(* CODESYS project mobject-graph.library
   Company: mobject
   DefaultNamespace: mobject-graph
   Version: 0.1.0
   Placeholder: mobject-graph
   Author: mobject dev team
   Title: mobject-graph

Project tree, tasks and I/O mapping:
  libraries: mobject-collections, 1.1.0 (mobject); mobject-datatypes, 0.4.1 (mobject); mobject-deserialization, 0.1.0 (mobject); mobject-disposable, 1.0.0 (mobject); mobject-enumerable, 1.1.0 (mobject); mobject-errors, 0.2.0 (mobject); mobject-events, 1.0.0 (mobject); mobject-serialization, 0.4.0 (mobject); Tc2_Standard, * (Beckhoff Automation GmbH); Tc2_System, * (Beckhoff Automation GmbH); Tc2_Utilities, * (Beckhoff Automation GmbH)
  Alarms/
    Base/
      function block Alarm [ST]: Active, Clear, Message, Reason, FB_init, Accept, RegisterWithParent, SerializeWith
    Events/
      function block AlarmAddedEvent [ST]: FB_init, Target
      interface I_AlarmAddedEvent: Target
    Host/
      function block AlarmHost [ST]: FB_init, EmitOnAlarmAddedEvent, Accept, AddAlarm, HasAlarms, HasRaisedAlarm, SerializeWith
    Interfaces/
      interface I_Alarm: Accept, Active, Message, Reason
      interface I_Alarms: Accept, AddAlarm, HasAlarms, HasRaisedAlarm
      interface I_HostAlarms: Alarms
    function block DeserializationFailedAlarm [ST]: Active, Clear, Message, Raise, Reason
    function block DeserializationFailedNodeNotSupportedAlarm [ST]: Active, Clear, Message, Raise, Reason
    function block FunctionFailedAlarm [ST]: Active, Clear, Message, Raise, Reason
  Content/
    Base/
      function block Content [ST]: FB_init, Accept, AddMetadata, Data, Metadatum, Name, OffEvent, OnceEvent, OnEvent, Parent, RegisterWithParent, SerializeWith
    Events/
      function block ContentAddedEvent [ST]: FB_init, Target
      interface I_ContentAddedEvent: Target
    Host/
      function block ContentHost [ST]: FB_init, FB_exit, CreateContent, DisposeSelfCreatedContent, EmitOnContentAddedEvent, Accept, AddContent, AddDataAsContent, HasContents, SerializeWith, TryGetContentByName
    Interface/
      interface I_Content: Accept, Data, Name, Parent
      interface I_Contents: Accept, AddContent, AddDataAsContent, HasContents, TryGetContentByName
      interface I_HostContent: Contents
  Errors/
    function block MissingNodePrototypeDeserializationError [ST]: FB_init, ErrorType, Message
  Extensions/
    Base/
      function block Extension [ST]: FB_init, Accept, AddMetadata, Alarms, Contents, HasRaisedAlarm, InputPorts, Metadatum, Name, OffEvent, OnceEvent, OnEvent, OutputPorts, Parameters, SerializeWith, TryDeserializeFrom
    Events/
      function block ExtensionAddedEvent [ST]: FB_init, Target
      interface I_ExtensionAddedEvent: Target
    Host/
      function block ExtensionHost [ST]: FB_init, EmitOnExtensionAddedEvent, Accept, AddExtension, HasExtensions, SerializeWith, TryDeserializeFrom, TryGetExtensionByName
    Interface/
      interface I_Extension: Accept, Name
      interface I_Extensions: Accept, AddExtension, HasExtensions, TryGetExtensionByName
      interface I_HostExtensions: Extensions
    Namespace/
      function block ExtensionNamespace [ST]: FB_init, ExtensionName, Initialize, IsExtensionPath, TargetName
  Graph/
    Base/
      function block Graph [ST]: FB_init, FB_exit, DisposeSelfCreatedNodes, TryDeserializeLinks, TryDeserializeNodes, Accept, AddMetadata, Alarms, Contents, Execute, Extensions, HasRaisedAlarm, InputPorts, Metadatum, Nodes, OffEvent, OnceEvent, OnEvent, OutputPorts, Parameters, Reset, SerializeWith, TryDeserializeFrom, Uuid
    Events/
      function block GraphAddedEvent [ST]: FB_init, Target
      interface I_GraphAddedEvent: Target
    Host/
      function block GraphHost [ST]: FB_init, EmitOnGraphAddedEvent, Accept, AddGraph, DisposeAll, Execute, RemoveGraph, SerializeWith, TryGetGraphByUuid
    Interfaces/
      interface I_Graph: Accept, Execute, Reset, Uuid
      interface I_Graphs: Accept, AddGraph, DisposeAll, Execute, RemoveGraph, TryGetGraphByUuid
      interface I_HostGraphs: Graphs
  GraphFramework/
    Interface/
      interface I_GraphFramework: Create, Datatypes, NodeFactory
    function block GraphFramework [ST]: Create, Datatypes, InstallDatatypePack, InstallNodePack, NodeFactory
  InputPort/
    Base/
      function block InputPort [ST]: FB_init, EmitOnInputPortChanged, HandleOutputPortChangedEvent, Accept, AddMetadata, Connected, Data, Disconnect, HandleEvent, Metadatum, Name, OffEvent, OnceEvent, OnEvent, RegisterWithParent, SerializeWith, TryConnectTo
    Events/
      interface I_InputPortAddedEvent: Target
      interface I_InputPortChangedEvent: Target
      function block InputPortAddedEvent [ST]: FB_init, Target
      function block InputPortChangedEvent [ST]: FB_init, Target
    Host/
      function block InputPortHost [ST]: FB_init, FB_exit, CreateInputPort, DisposeSelfCreatedInputPorts, EmitOnPortAddedEvent, Accept, AddDataAsInputPort, AddInputPort, HasInputPorts, SerializeWith, TryGetInputPortByName
    Interface/
      interface I_HostInputPorts: InputPorts
      interface I_InputPort: Accept, Connected, Data, Disconnect, Name, TryConnectTo
      interface I_InputPorts: Accept, AddDataAsInputPort, AddInputPort, HasInputPorts, TryGetInputPortByName
  Metadata/
    Base/
      function block Metadata [ST]: FB_init, Accept, Data, Name, Parent, RegisterWithParent, SerializeWith
    Events/
      interface I_MetadataAddedEvent: Target
      function block MetadataAddedEvent [ST]: FB_init, Target
    Host/
      function block MetadataHost [ST]: FB_init, FB_exit, CreateMetadata, DisposeSelfCreatedMetadata, EmitOnMetadataAddedEvent, Accept, AddDataAsMetadata, AddMetadata, HasMetadata, SerializeWith, TryGetMetadataByName
    Interface/
      interface I_HostMetadata: AddMetadata, Metadatum
      interface I_Metadata: Accept, Data, Name, SerializeWith
      interface I_Metadatum: Accept, AddDataAsMetadata, AddMetadata, HasMetadata, TryGetMetadataByName
  Node/
    Base/
      function block Node [ST]: Clone, OnExecute, EmitNodeExecuteBeginEvent, EmitNodeExecuteEndEvent, EmitOnNodePreExecuteEvent, AddContent, AddInput, AddOutput, AddParameter, Accept, AddMetadata, Alarms, Contents, Execute, Extensions, HasRaisedAlarm, Id, InputPorts, Metadatum, Mode, OffEvent, OnceEvent, OnEvent, Order, OutputPorts, Parameters, Self, SerializeWith, TryDeserializeFrom
    Events/
      interface I_NodeAddedEvent: Target
      interface I_NodeExecuteBeginEvent: Target
      interface I_NodeExecuteEndEvent: Target
      interface I_NodePreExecuteEvent: Cancel, ExecuteCancelled, Target
      function block NodeAddedEvent [ST]: FB_init, Target
      function block NodeExecuteBeginEvent [ST]: FB_init, CpuCounterHighBytes, CpuCounterLowBytes, Target
      function block NodeExecuteEndEvent [ST]: FB_init, CpuCounterHighBytes, CpuCounterLowBytes, Target
      function block NodePreExecuteEvent [ST]: FB_init, Cancel, ExecuteCancelled, Target
    Host/
      function block NodeHost [ST]: FB_init, EmitOnNodeAddedEvent, UpdateExecutionOrder, Accept, AddNode, Execute, HasNodes, RemoveNode, SerializeWith, TryDeserializeFrom, TryGetNodeById
    Interface/
      interface I_HostNodes: Nodes
      interface I_Node: Accept, Clone, Execute, Id, Mode, Order
      interface I_Nodes: Accept, AddNode, HasNodes, TryGetNodeById
  NodeFactory/
    Base/
      function block NodeFactory [ST]: Accept, AddNodeAsPrototype, AddNodePrototype, NodePrototypes, TryCreateNodeByType
    Interface/
      interface I_NodeFactory: Accept, AddNodeAsPrototype, AddNodePrototype, NodePrototypes, TryCreateNodeByType
  NodePack/
    interface I_NodePack: RegisterWithNodeFactory
  NodePrototype/
    Base/
      function block NodePrototype [ST]: FB_init, Accept, Clone, Node, Path
    Host/
      function block NodePrototypeHost [ST]: FB_exit, CreatePrototype, DisposeSelfCreatedNodePrototypes, Accept, AddNodeAsPrototype, AddNodePrototype, HasNodePrototypes, TryGetNodePrototypeByPath
    Interface/
      interface I_NodePrototype: Accept, Clone, Node, Path
      interface I_NodePrototypes: Accept, HasNodePrototypes
  OutputPort/
    Base/
      function block OutputPort [ST]: FB_init, EmitOnOutputPortChangeEvent, Accept, AddMetadata, Data, Metadatum, Name, OffEvent, OnceEvent, OnEvent, RegisterWithParent, SerializeWith
    Events/
      interface I_OutputPortAddedEvent: Target
      interface I_OutputPortChangedEvent: Target
      function block OutputPortAddedEvent [ST]: FB_init, Target
      function block OutputPortChangedEvent [ST]: FB_init, Target
    Host/
      function block OutputPortHost [ST]: FB_init, FB_exit, CreateOutputPort, DisposeSelfCreatedOutputPorts, EmitOnPortAddedEvent, Accept, AddDataAsOutputPort, AddOutputPort, HasOutputPorts, SerializeWith, TryGetOutputPortByName
    Interface/
      interface I_HostOutputPorts: OutputPorts
      interface I_OutputPort: Accept, Data, Name
      interface I_OutputPorts: Accept, AddDataAsOutputPort, AddOutputPort, HasOutputPorts, TryGetOutputPortByName
  Parameters/
    Base/
      function block Parameter [ST]: FB_init, Accept, AddMetadata, Data, Metadatum, Name, OffEvent, OnceEvent, OnEvent, Parent, RegisterWithParent, SerializeWith, TryDeserializeFrom
    Events/
      interface I_ParameterAddedEvent: TargetParameter
      function block ParameterAddedEvent [ST]: FB_init, TargetParameter
    Host/
      function block ParameterHost [ST]: FB_init, FB_exit, CreateParameter, DisposeSelfCreatedParameters, EmitOnParameterAddedEvent, Accept, AddDataAsParameter, AddParameter, HasParameters, SerializeWith, TryDeserializeFrom, TryGetParameterByName
    Interface/
      interface I_HostParameters: Parameters
      interface I_Parameter: Accept, Data, Name, Parent
      interface I_Parameters: Accept, AddDataAsParameter, AddParameter, HasParameters, TryGetParameterByName
  Visitors/
    Interfaces/
      interface I_AlarmVisitor: VisitAlarm
      interface I_ContentVisitor: VisitContent
      interface I_ExtensionVisitor: VisitExtension
      interface I_GraphVisitor: VisitGraph
      interface I_InputPortVisitor: VisitInputPort
      interface I_MetadataVisitor: VisitMetadatum
      interface I_NodeFactoryVisitor: VisitNodeFactory
      interface I_NodePrototypeVisitor: VisitNodePrototype
      interface I_NodeVisitor: VisitNode
      interface I_OutputPortVisitor: VisitOutputPort
      interface I_ParameterVisitor: VisitParameter
*)

// Alarms/Base/Alarm
{attribute 'linkalways'} 
{attribute 'no_explicit_call' := 'This FB is a CLASS and must be accessed using methods or properties'}
{attribute 'enable_dynamic_creation'}
FUNCTION_BLOCK ABSTRACT Alarm IMPLEMENTS I_Alarm

PROPERTY ABSTRACT Active : BOOL
GET
END_GET
END_PROPERTY

METHOD ABSTRACT Clear
END_METHOD

PROPERTY ABSTRACT Message : T_MaxString
GET
END_GET
END_PROPERTY

PROPERTY ABSTRACT Reason : T_MaxString
GET
END_GET
END_PROPERTY

METHOD FB_init : BOOL
VAR_INPUT
	bInitRetains : BOOL; // if TRUE, the retain variables are initialized (warm start / cold start)
	bInCopyCode : BOOL;  // if TRUE, the instance afterwards gets moved into the copy code (online change)
	Parent : I_HostAlarms;
END_VAR
RegisterWithParent(Parent);
END_METHOD

METHOD PUBLIC Accept
VAR_INPUT
	Visitor : I_AlarmVisitor;
END_VAR
Visitor.VisitAlarm(this^);
END_METHOD

METHOD RegisterWithParent
VAR_INPUT
	Parent : I_HostAlarms;
END_VAR
IF Parent = 0 THEN
	RETURN;
END_IF

Parent.Alarms.AddAlarm(THIS^);
END_METHOD

METHOD PUBLIC SerializeWith
VAR_INPUT
	Serializer : I_Serializer;
END_VAR
VAR
	isActive : BOOL := Active;
	errorMessage : T_MAXSTRING := Message;
	reasonMessage : T_MAXSTRING := Reason;
END_VAR
Serializer.StartObject();
Serializer.AddKeyString('message',errorMessage);
Serializer.AddKeyBool('active',isActive);

IF reasonMessage <> '' THEN
	Serializer.AddKeyString('reason',reasonMessage);
END_IF

Serializer.EndObject();
END_METHOD

END_FUNCTION_BLOCK

// Alarms/Interfaces/I_Alarm
INTERFACE I_Alarm EXTENDS I_Serializable

METHOD PUBLIC Accept
VAR_INPUT
	Visitor : I_AlarmVisitor;
END_VAR
END_METHOD

PROPERTY PUBLIC Active : BOOL
GET
END_GET
END_PROPERTY

PROPERTY PUBLIC Message : T_MaxString
GET
END_GET
END_PROPERTY

PROPERTY PUBLIC Reason : T_MaxString
GET
END_GET
END_PROPERTY

END_INTERFACE

// Visitors/Interfaces/I_AlarmVisitor
INTERFACE I_AlarmVisitor

METHOD VisitAlarm
VAR_INPUT
	VisitingAlarm : I_Alarm;
END_VAR
END_METHOD

END_INTERFACE

// Alarms/Interfaces/I_HostAlarms
INTERFACE I_HostAlarms EXTENDS __SYSTEM.IQueryInterface

PROPERTY Alarms : I_Alarms
GET
END_GET
END_PROPERTY

END_INTERFACE

// Alarms/Interfaces/I_Alarms
INTERFACE I_Alarms

METHOD PUBLIC Accept
VAR_INPUT
	Visitor : I_AlarmVisitor;
END_VAR
END_METHOD

METHOD AddAlarm
VAR_INPUT
	Alarm : I_Alarm;
END_VAR
END_METHOD

PROPERTY PUBLIC HasAlarms : BOOL
GET
END_GET
END_PROPERTY

PROPERTY PUBLIC HasRaisedAlarm : BOOL
GET
END_GET
END_PROPERTY

END_INTERFACE

// Alarms/Events/AlarmAddedEvent
{attribute 'linkalways'} 
{attribute 'no_explicit_call' := 'This FB is a CLASS and must be accessed using methods or properties'}
{attribute 'enable_dynamic_creation'}
FUNCTION_BLOCK AlarmAddedEvent EXTENDS Disposable IMPLEMENTS I_AlarmAddedEvent
VAR
	_target : I_Alarm;
END_VAR

METHOD FB_init : BOOL
VAR_INPUT
	bInitRetains : BOOL; // if TRUE, the retain variables are initialized (warm start / cold start)
	bInCopyCode : BOOL;  // if TRUE, the instance afterwards gets moved into the copy code (online change)
	Target : I_Alarm;
END_VAR
This^._target := Target;
END_METHOD

PROPERTY PUBLIC Target : I_Alarm
GET
Target := _target;
END_GET
END_PROPERTY

END_FUNCTION_BLOCK

// Alarms/Events/I_AlarmAddedEvent
INTERFACE I_AlarmAddedEvent EXTENDS I_Event

PROPERTY PUBLIC Target : I_Alarm
GET
END_GET
END_PROPERTY

END_INTERFACE

// Alarms/Host/AlarmHost
{attribute 'linkalways'} 
{attribute 'no_explicit_call' := 'This FB is a CLASS and must be accessed using methods or properties'}
{attribute 'enable_dynamic_creation'}
FUNCTION_BLOCK AlarmHost IMPLEMENTS I_Alarms, I_Serializable
VAR
	hostParent : I_HostAlarms;
	eventTarget : I_EventTarget;
	alarms : Stack;
END_VAR

METHOD FB_init : BOOL
VAR_INPUT
	bInitRetains : BOOL; // if TRUE, the retain variables are initialized (warm start / cold start)
	bInCopyCode : BOOL;  // if TRUE, the instance afterwards gets moved into the copy code (online change)
	Parent : I_HostAlarms;
	ParentEventTarget : I_EventTarget;
END_VAR
hostParent := Parent;
eventTarget := parentEventTarget;
END_METHOD

METHOD PROTECTED EmitOnAlarmAddedEvent
VAR_INPUT
	Alarm : I_Alarm;
END_VAR
VAR
	pAlarmAddedEvent : POINTER TO AlarmAddedEvent;
END_VAR
IF eventTarget = 0 THEN
	RETURN;
END_IF

pAlarmAddedEvent := __NEW(AlarmAddedEvent(Target := Alarm));
eventTarget.Emit('OnAlarmAdded',pAlarmAddedEvent^);
pAlarmAddedEvent^.Dispose();
END_METHOD

METHOD PUBLIC Accept
VAR_INPUT
	Visitor : I_AlarmVisitor;
END_VAR
VAR
	enumerator : I_ForwardEnumerator;
	alarm : I_Alarm;
END_VAR
enumerator := alarms.GetEnumerator();

WHILE (enumerator.MoveNext()) DO
	
	IF enumerator.TryGet(alarm) THEN
		alarm.Accept(Visitor);
	END_IF

END_WHILE

enumerator.Dispose();
END_METHOD

METHOD PUBLIC AddAlarm
VAR_INPUT
	Alarm : I_Alarm;
END_VAR
alarms.Push(Alarm);
EmitOnAlarmAddedEvent(Alarm);
END_METHOD

PROPERTY PUBLIC HasAlarms : BOOL
GET
HasAlarms := alarms.Count > 0;
END_GET
END_PROPERTY

PROPERTY PUBLIC HasRaisedAlarm : BOOL
GET
VAR
	enumerator : I_ForwardEnumerator;
	alarm : I_Alarm;
END_VAR
enumerator := alarms.GetEnumerator();

WHILE (enumerator.MoveNext()) DO
	
	IF NOT enumerator.TryGet(alarm) THEN
		CONTINUE;
	END_IF
	
	IF alarm.Active THEN
		HasRaisedAlarm := TRUE;
		EXIT;
	END_IF

END_WHILE

enumerator.Dispose();
END_GET
END_PROPERTY

METHOD PUBLIC SerializeWith
VAR_INPUT
	Serializer : I_Serializer;
END_VAR
VAR
	enumerator : I_ForwardEnumerator;
	alarm : I_Alarm;
END_VAR
IF alarms.Count = 0 THEN
	RETURN;
END_IF

Serializer.AddKey('alarms');
Serializer.StartArray();

enumerator := alarms.GetEnumerator();

WHILE enumerator.MoveNext() DO
	IF enumerator.TryGet(alarm) THEN
		alarm.SerializeWith(Serializer);
	END_IF
END_WHILE

Serializer.EndArray();
enumerator.Dispose();
END_METHOD

END_FUNCTION_BLOCK

// Alarms/DeserializationFailedAlarm
{attribute 'linkalways'} 
{attribute 'no_explicit_call' := 'This FB is a CLASS and must be accessed using methods or properties'}
{attribute 'enable_dynamic_creation'}
FUNCTION_BLOCK PUBLIC DeserializationFailedAlarm EXTENDS Alarm
VAR
	state : (CLEARED, RAISED);
	_reason : T_MAXSTRING;
END_VAR

PROPERTY Active : BOOL
GET
Active := state <> CLEARED;
END_GET
END_PROPERTY

METHOD PUBLIC Clear
_reason := '';
state := CLEARED;
END_METHOD

PROPERTY PUBLIC Message : T_MaxString
GET
Message := 'Deserialization failed';
END_GET
END_PROPERTY

METHOD PUBLIC Raise
VAR_INPUT
	Reason : T_MAXSTRING;
END_VAR
_reason := Reason;
state := RAISED;
END_METHOD

PROPERTY Reason : T_MaxString
GET
Reason := _reason;
END_GET
END_PROPERTY

END_FUNCTION_BLOCK

// Alarms/DeserializationFailedNodeNotSupportedAlarm
{attribute 'linkalways'} 
{attribute 'no_explicit_call' := 'This FB is a CLASS and must be accessed using methods or properties'}
{attribute 'enable_dynamic_creation'}
FUNCTION_BLOCK PUBLIC DeserializationFailedNodeNotSupportedAlarm EXTENDS Alarm
VAR
	state : (CLEARED, RAISED);
	_reason : T_MAXSTRING;
END_VAR

PROPERTY Active : BOOL
GET
Active := state <> CLEARED;
END_GET
END_PROPERTY

METHOD PUBLIC Clear
_reason := '';
state := CLEARED;
END_METHOD

PROPERTY PUBLIC Message : T_MaxString
GET
Message := 'Node type is not installed';
END_GET
END_PROPERTY

METHOD PUBLIC Raise
VAR_INPUT
	NodeType : T_MAXSTRING;
END_VAR
_reason := NodeType;
state := RAISED;
END_METHOD

PROPERTY Reason : T_MaxString
GET
Reason := _reason;
END_GET
END_PROPERTY

END_FUNCTION_BLOCK

// Node/Base/Node
{attribute 'linkalways'} 
{attribute 'no_explicit_call' := 'This FB is a CLASS and must be accessed using methods or properties'}
{attribute 'enable_dynamic_creation'}
FUNCTION_BLOCK ABSTRACT Node EXTENDS Disposable IMPLEMENTS I_Node
VAR
	_id : T_MAXSTRING;
	_order : DINT;
	_mode : DINT;
	eventEmitter : EventEmitter;
	inputPortHost : InputPortHost(THIS^, eventEmitter);
	outputPortHost : OutputPortHost(THIS^, eventEmitter);
	parameterHost : ParameterHost(THIS^, eventEmitter);
	contentHost : ContentHost(THIS^, eventEmitter);
	alarmHost : AlarmHost(THIS^, eventEmitter);
	metadataHost : MetadataHost(THIS^, eventEmitter);
	extensionHost : ExtensionHost(THIS^,eventEmitter);
	deserializationFailedAlarm : DeserializationFailedAlarm(THIS^);
END_VAR

METHOD PUBLIC ABSTRACT Clone : I_Node
VAR_INPUT
END_VAR
END_METHOD

METHOD PROTECTED ABSTRACT OnExecute : HRESULT
END_METHOD

METHOD PRIVATE EmitNodeExecuteBeginEvent : BOOL;
VAR
	pNodeExecuteBeginEvent : POINTER TO NodeExecuteBeginEvent;
END_VAR
pNodeExecuteBeginEvent := __NEW(NodeExecuteBeginEvent(Target := THIS^));
eventEmitter.Emit('OnNodeExecuteBegin',pNodeExecuteBeginEvent^);
pNodeExecuteBeginEvent^.Dispose();
END_METHOD

METHOD PRIVATE EmitNodeExecuteEndEvent : BOOL;
VAR
	pNodeExecuteEndEvent : POINTER TO NodeExecuteEndEvent;
END_VAR
pNodeExecuteEndEvent := __NEW(NodeExecuteEndEvent(Target := THIS^));
eventEmitter.Emit('OnNodeExecuteEnd',pNodeExecuteEndEvent^);
pNodeExecuteEndEvent^.Dispose();
END_METHOD

METHOD PRIVATE EmitOnNodePreExecuteEvent : BOOL;
VAR_INPUT
	CancelRequested : REFERENCE TO BOOL;
END_VAR
VAR
	pNodePreExecuteEvent : POINTER TO NodePreExecuteEvent;
END_VAR
pNodePreExecuteEvent := __NEW(NodePreExecuteEvent(Target := THIS^));
eventEmitter.Emit('OnNodePreExecute',pNodePreExecuteEvent^);

IF pNodePreExecuteEvent^.ExecuteCancelled THEN
	CancelRequested := TRUE;
END_IF

pNodePreExecuteEvent^.Dispose();
END_METHOD

METHOD PROTECTED AddContent : I_Content
VAR_INPUT
	Name : T_MAXSTRING;
	Data : I_Datatype;
END_VAR
AddContent := Contents.AddDataAsContent(Name, Data);
END_METHOD

METHOD PROTECTED AddInput : I_InputPort
VAR_INPUT
	Name : T_MAXSTRING;
	Data : I_Datatype;
END_VAR
AddInput := InputPorts.AddDataAsInputPort(Name, Data);
END_METHOD

METHOD PROTECTED AddOutput : I_OutputPort
VAR_INPUT
	Name : T_MAXSTRING;
	Data : I_Datatype;
END_VAR
AddOutput := OutputPorts.AddDataAsOutputPort(Name, Data);
END_METHOD

METHOD PROTECTED AddParameter : I_Parameter
VAR_INPUT
	Name : T_MAXSTRING;
	Data : I_Datatype;
END_VAR
AddParameter := Parameters.AddDataAsParameter(Name, Data);
END_METHOD

METHOD PUBLIC Accept
VAR_INPUT
	Visitor : I_NodeVisitor;
END_VAR
Visitor.VisitNode(THIS^);
END_METHOD

METHOD PUBLIC AddMetadata : I_HostMetadata
VAR_INPUT
	Name : T_MAXSTRING;
	Data : I_Datatype;
END_VAR
Metadatum.AddDataAsMetadata(Name, Data);
AddMetadata := THIS^;
END_METHOD

PROPERTY PUBLIC Alarms : I_Alarms
GET
Alarms := alarmHost;
END_GET
END_PROPERTY

PROPERTY PUBLIC Contents : I_Contents
GET
Contents := contentHost;
END_GET
END_PROPERTY

METHOD PUBLIC Execute
VAR
	cancelExecuteResponse : BOOL := FALSE;
END_VAR
EmitOnNodePreExecuteEvent(cancelExecuteResponse);

IF cancelExecuteResponse THEN
	RETURN;
END_IF

EmitNodeExecuteBeginEvent();
OnExecute();
EmitNodeExecuteEndEvent();
END_METHOD

PROPERTY PUBLIC Extensions : I_Extensions
GET
Extensions := extensionHost;
END_GET
END_PROPERTY

PROPERTY PUBLIC HasRaisedAlarm : BOOL
GET
HasRaisedAlarm := alarmHost.HasRaisedAlarm;
END_GET
END_PROPERTY

PROPERTY PUBLIC Id : T_MAXSTRING
GET
Id := _id;
END_GET
END_PROPERTY

PROPERTY PUBLIC InputPorts : I_InputPorts
GET
InputPorts := inputPortHost;
END_GET
END_PROPERTY

PROPERTY PUBLIC Metadatum : I_Metadatum
GET
Metadatum := metadataHost;
END_GET
END_PROPERTY

PROPERTY PUBLIC Mode : DINT
GET
Mode := _mode;
END_GET
END_PROPERTY

METHOD PUBLIC OffEvent
VAR_INPUT
	EventName : T_MaxString;
	EventHandler : I_EventHandler;
END_VAR
eventEmitter.OffEvent(EventName, EventHandler);
END_METHOD

METHOD PUBLIC OnceEvent
VAR_INPUT
	EventName : T_MaxString;
	EventHandler : I_EventHandler;
END_VAR
eventEmitter.OnceEvent(EventName, EventHandler);
END_METHOD

METHOD PUBLIC OnEvent
VAR_INPUT
	EventName : T_MaxString;
	EventHandler : I_EventHandler;
END_VAR
eventEmitter.OnEvent(EventName, EventHandler);
END_METHOD

PROPERTY PUBLIC Order : DINT
GET
Order := _order;
END_GET
END_PROPERTY

PROPERTY PUBLIC OutputPorts : I_OutputPorts
GET
OutputPorts := outputPortHost;
END_GET
END_PROPERTY

PROPERTY PUBLIC Parameters : I_Parameters
GET
Parameters := parameterHost;
END_GET
END_PROPERTY

PROPERTY PUBLIC Self : I_Node
GET
Self := This^;
END_GET
END_PROPERTY

METHOD PUBLIC SerializeWith
VAR_INPUT
	Serializer : I_Serializer;
END_VAR
Serializer.StartObject();
Serializer.AddKeyString('id',_id);
Serializer.AddKeyDint('order',_order);
Serializer.AddKeyDint('mode',_mode);
inputPortHost.SerializeWith(Serializer);
outputPortHost.SerializeWith(Serializer);
parameterHost.SerializeWith(Serializer);
contentHost.SerializeWith(Serializer);
alarmHost.SerializeWith(Serializer);
extensionHost.SerializeWith(Serializer);
metadataHost.SerializeWith(Serializer);
Serializer.EndObject();
END_METHOD

METHOD PUBLIC TryDeserializeFrom : BOOL
VAR_INPUT
	Deserializer : I_Deserializer;
	Feedback : I_DeserializerFeedback;
END_VAR
DeserializationFailedAlarm.Clear();

IF NOT Deserializer.TryGetKeyString('id', _id, Feedback) THEN
	DeserializationFailedAlarm.Raise('Missing node id');	
	RETURN;
END_IF

IF NOT Deserializer.TryGetKeyDint('order', _order, Feedback) THEN
	DeserializationFailedAlarm.Raise('Missing node order');	
	RETURN;
END_IF

IF NOT Deserializer.TryGetKeyDint('mode', _mode, Feedback) THEN
	DeserializationFailedAlarm.Raise('Missing node mode');	
	RETURN;
END_IF

IF NOT parameterHost.TryDeserializeFrom(Deserializer, Feedback) THEN
	DeserializationFailedAlarm.Raise('Failed to deserialize parameters');	
	RETURN;
END_IF

IF NOT extensionHost.TryDeserializeFrom(Deserializer, Feedback) THEN
	DeserializationFailedAlarm.Raise('Failed to deserialize extensions');	
	RETURN;
END_IF

TryDeserializeFrom := TRUE;
END_METHOD

END_FUNCTION_BLOCK

// Node/Interface/I_Node
INTERFACE I_Node EXTENDS I_Disposable, I_HostContent, I_HostInputPorts, I_HostOutputPorts, I_HostAlarms, I_HostParameters, I_HostExtensions, I_HostMetadata, I_EventEmitter, I_Deserializable, I_Serializable

METHOD PUBLIC Accept
VAR_INPUT
	Visitor : I_NodeVisitor;
END_VAR
END_METHOD

METHOD Clone : I_Node
VAR_INPUT
END_VAR
END_METHOD

METHOD PUBLIC Execute
END_METHOD

PROPERTY PUBLIC Id : T_MAXSTRING
GET
END_GET
END_PROPERTY

PROPERTY PUBLIC Mode : DINT
GET
END_GET
END_PROPERTY

PROPERTY PUBLIC Order : DINT
GET
END_GET
END_PROPERTY

END_INTERFACE

// Content/Interface/I_HostContent
INTERFACE I_HostContent

PROPERTY PUBLIC Contents : I_Contents
GET
END_GET
END_PROPERTY

END_INTERFACE

// Content/Interface/I_Contents
INTERFACE I_Contents

METHOD PUBLIC Accept
VAR_INPUT
	visitor : I_ContentVisitor;
END_VAR
END_METHOD

METHOD AddContent
VAR_INPUT
	Content : I_Content;
END_VAR
END_METHOD

METHOD PUBLIC AddDataAsContent : I_Content
VAR_INPUT
	Name : T_MAXSTRING;
	Data : I_Datatype;
END_VAR
END_METHOD

PROPERTY PUBLIC HasContents : BOOL
GET
END_GET
END_PROPERTY

METHOD PUBLIC TryGetContentByName : BOOL
VAR_INPUT
	Name : T_MAXSTRING;
	Destination : REFERENCE TO I_Content;
END_VAR
END_METHOD

END_INTERFACE

// Visitors/Interfaces/I_ContentVisitor
INTERFACE I_ContentVisitor

METHOD VisitContent
VAR_INPUT
	VisitingContent : I_Content;
END_VAR
END_METHOD

END_INTERFACE

// Content/Interface/I_Content
INTERFACE I_Content EXTENDS I_Disposable, I_Serializable, I_HostMetadata, I_EventEmitter

METHOD PUBLIC Accept
VAR_INPUT
	Visitor : I_ContentVisitor;
END_VAR
END_METHOD

PROPERTY PUBLIC Data : I_DataType
GET
END_GET
END_PROPERTY

PROPERTY PUBLIC Name : T_MAXSTRING
GET
END_GET
END_PROPERTY

PROPERTY PUBLIC Parent : I_HostContent
GET
END_GET
END_PROPERTY

END_INTERFACE

// Metadata/Interface/I_HostMetadata
INTERFACE I_HostMetadata EXTENDS __SYSTEM.IQueryInterface

METHOD PUBLIC AddMetadata : I_HostMetadata
VAR_INPUT
	Name : T_MAXSTRING;
	Data : I_Datatype;
END_VAR
END_METHOD

PROPERTY Metadatum : I_Metadatum
GET
END_GET
END_PROPERTY

END_INTERFACE

// Metadata/Interface/I_Metadatum
INTERFACE I_Metadatum

METHOD PUBLIC Accept
VAR_INPUT
	Visitor : I_MetadataVisitor;
END_VAR
END_METHOD

METHOD PUBLIC AddDataAsMetadata : I_Metadata
VAR_INPUT
	Name : T_MAXSTRING;
	Data : I_Datatype;
END_VAR
END_METHOD

METHOD AddMetadata
VAR_INPUT
	Metadata : I_Metadata;
END_VAR
END_METHOD

PROPERTY PUBLIC HasMetadata : BOOL
GET
END_GET
END_PROPERTY

METHOD PUBLIC TryGetMetadataByName : BOOL
VAR_INPUT
	Name : T_MAXSTRING;
	Destination : REFERENCE TO I_Metadata;
END_VAR
END_METHOD

END_INTERFACE

// Visitors/Interfaces/I_MetadataVisitor
INTERFACE I_MetadataVisitor

METHOD VisitMetadatum
VAR_INPUT
	VisitingMetadatum : I_Metadata;
END_VAR
END_METHOD

END_INTERFACE

// Metadata/Interface/I_Metadata
INTERFACE I_Metadata EXTENDS I_Disposable, I_Serializable

METHOD PUBLIC Accept
VAR_INPUT
	Visitor : I_MetadataVisitor;
END_VAR
END_METHOD

PROPERTY PUBLIC Data : I_DataType
GET
END_GET
END_PROPERTY

PROPERTY PUBLIC Name : T_MAXSTRING
GET
END_GET
END_PROPERTY

METHOD PUBLIC SerializeWith
VAR_INPUT
	Serializer : I_Serializer;
END_VAR
END_METHOD

END_INTERFACE

// Metadata/Base/Metadata
{attribute 'linkalways'} 
{attribute 'no_explicit_call' := 'This FB is a CLASS and must be accessed using methods or properties'}
{attribute 'enable_dynamic_creation'}
FUNCTION_BLOCK Metadata EXTENDS Disposable IMPLEMENTS I_Metadata
VAR
	_name : T_MAXSTRING;
	_data : I_Datatype;
	_parent : I_HostMetadata;
END_VAR

METHOD FB_init : BOOL
VAR_INPUT
	bInitRetains : BOOL; // if TRUE, the retain variables are initialized (warm start / cold start)
	bInCopyCode : BOOL;  // if TRUE, the instance afterwards gets moved into the copy code (online change)
	Name : T_MAXSTRING;
	Data : I_Datatype;
	Parent : I_HostMetadata;
END_VAR
_name := Name;
_data := Data;
RegisterWithParent(Parent);
END_METHOD

METHOD PUBLIC Accept
VAR_INPUT
	Visitor : I_MetadataVisitor;
END_VAR
Visitor.VisitMetadatum(this^);
END_METHOD

PROPERTY PUBLIC Data : I_DataType
GET
Data := _data;
END_GET
END_PROPERTY

PROPERTY PUBLIC Name : T_MAXSTRING
GET
Name := _name;
END_GET
END_PROPERTY

PROPERTY PUBLIC Parent : I_HostMetadata
GET
Parent := _parent;
END_GET
END_PROPERTY

METHOD PUBLIC RegisterWithParent
VAR_INPUT
	Parent : I_HostMetadata;
END_VAR
IF Parent = 0 THEN
	RETURN;
END_IF

THIS^._parent := Parent;
Parent.Metadatum.AddMetadata(THIS^);
END_METHOD

METHOD PUBLIC SerializeWith
VAR_INPUT
	Serializer : I_Serializer;
END_VAR
Serializer.StartObject();
Serializer.AddKeyString('name',_name);
Serializer.Addkey('datatype');
_data.SerializeTypeWith(Serializer);
Serializer.AddkeyObject('value',_data);
Serializer.EndObject();
END_METHOD

END_FUNCTION_BLOCK

// Content/Base/Content
{attribute 'linkalways'} 
{attribute 'no_explicit_call' := 'This FB is a CLASS and must be accessed using methods or properties'}
{attribute 'enable_dynamic_creation'}
FUNCTION_BLOCK Content EXTENDS Disposable IMPLEMENTS I_Content
VAR
	_name : T_MAXSTRING;
	_data : I_Datatype;
	_parent : I_HostContent;
	eventEmitter : EventEmitter;
	metadataHost : MetadataHost(THIS^, eventEmitter);
END_VAR

METHOD FB_init : BOOL
VAR_INPUT
	bInitRetains : BOOL; // if TRUE, the retain variables are initialized (warm start / cold start)
	bInCopyCode : BOOL;  // if TRUE, the instance afterwards gets moved into the copy code (online change)
	Name : T_MAXSTRING;
	Data : I_Datatype;
	Parent : I_HostContent;
END_VAR
_name := Name;
_data := Data;
RegisterWithParent(Parent);
END_METHOD

METHOD PUBLIC Accept
VAR_INPUT
	Visitor : I_ContentVisitor;
END_VAR
Visitor.VisitContent(THIS^);
END_METHOD

METHOD PUBLIC AddMetadata : I_HostMetadata
VAR_INPUT
	Name : T_MAXSTRING;
	Data : I_Datatype;
END_VAR
Metadatum.AddDataAsMetadata(Name, Data);
AddMetadata := THIS^;
END_METHOD

PROPERTY PUBLIC Data : I_DataType
GET
Data := _data;
END_GET
END_PROPERTY

PROPERTY PUBLIC Metadatum : I_Metadatum
GET
Metadatum := metadataHost;
END_GET
END_PROPERTY

PROPERTY PUBLIC Name : T_MAXSTRING
GET
Name := _name;
END_GET
END_PROPERTY

METHOD PUBLIC OffEvent
VAR_INPUT
	EventName : T_MaxString;
	EventHandler : I_EventHandler;
END_VAR
eventEmitter.OffEvent(EventName, EventHandler);
END_METHOD

METHOD PUBLIC OnceEvent
VAR_INPUT
	EventName : T_MaxString;
	EventHandler : I_EventHandler;
END_VAR
eventEmitter.OnceEvent(EventName, EventHandler);
END_METHOD

METHOD PUBLIC OnEvent
VAR_INPUT
	EventName : T_MaxString;
	EventHandler : I_EventHandler;
END_VAR
eventEmitter.OnEvent(EventName, EventHandler);
END_METHOD

PROPERTY PUBLIC Parent : I_HostContent
GET
Parent := _parent;
END_GET
END_PROPERTY

METHOD PUBLIC RegisterWithParent
VAR_INPUT
	Parent : I_HostContent;
END_VAR
IF Parent = 0 THEN
	RETURN;
END_IF

THIS^._parent := Parent;
Parent.Contents.AddContent(THIS^);
END_METHOD

METHOD PUBLIC SerializeWith
VAR_INPUT
	Serializer : I_Serializer;
END_VAR
Serializer.StartObject();
Serializer.AddKeyString('name',_name);
Serializer.Addkey('datatype');
_data.SerializeTypeWith(Serializer);
Serializer.AddkeyObject('value',_data);
metadataHost.SerializeWith(Serializer);
Serializer.EndObject();
END_METHOD

END_FUNCTION_BLOCK

// Metadata/Host/MetadataHost
{attribute 'linkalways'} 
{attribute 'no_explicit_call' := 'This FB is a CLASS and must be accessed using methods or properties'}
{attribute 'enable_dynamic_creation'}
FUNCTION_BLOCK MetadataHost IMPLEMENTS I_Metadatum, I_Serializable
VAR
	hostParent : I_HostMetadata;
	eventTarget : I_EventTarget;
	meta : Dictionary;
	selfCreatedMetadata : Stack;
END_VAR

METHOD FB_init : BOOL
VAR_INPUT
	bInitRetains : BOOL; // if TRUE, the retain variables are initialized (warm start / cold start)
	bInCopyCode : BOOL;  // if TRUE, the instance afterwards gets moved into the copy code (online change)
	Parent : I_HostMetadata;
	ParentEventTarget : I_EventTarget;
END_VAR
hostParent := Parent;
eventTarget := ParentEventTarget;
END_METHOD

METHOD FB_exit : BOOL
VAR_INPUT
	bInCopyCode : BOOL; // if TRUE, the exit method is called for exiting an instance that is copied afterwards (online change).
END_VAR
IF bInCopyCode THEN
	RETURN;
END_IF

DisposeSelfCreatedMetadata();
END_METHOD

METHOD PRIVATE CreateMetadata : I_Metadata
VAR_INPUT
	MetadataName : T_MAXSTRING;
	MetadataData : I_Datatype;
END_VAR
VAR
	pMetadata : POINTER TO Metadata;
END_VAR
pMetadata := __NEW(Metadata(Name := MetadataName, Data := MetadataData, Parent := hostParent));
CreateMetadata := pMetadata^;
END_METHOD

METHOD PROTECTED DisposeSelfCreatedMetadata : BOOL
VAR
	metadata : I_Metadata;
END_VAR
WHILE selfCreatedMetadata.TryPop(metadata) DO
	metadata.Dispose();
END_WHILE
END_METHOD

METHOD PROTECTED EmitOnMetadataAddedEvent
VAR_INPUT
	Metadata : I_Metadata;
END_VAR
VAR
	pMetadataAddedEvent : POINTER TO MetadataAddedEvent;
END_VAR
IF eventTarget = 0 THEN
	RETURN;
END_IF

pMetadataAddedEvent := __NEW(MetadataAddedEvent(Target := Metadata));
eventTarget.Emit('OnMetadataAdded',pMetadataAddedEvent^);
pMetadataAddedEvent^.Dispose();
END_METHOD

METHOD PUBLIC Accept
VAR_INPUT
	Visitor : I_MetadataVisitor;
END_VAR
VAR
	enumerator : I_ForwardEnumerator;
	metadata : I_Metadata;
END_VAR
enumerator := meta.GetEnumerator();

WHILE (enumerator.MoveNext()) DO
	
	IF enumerator.TryGet(metadata) THEN
		metadata.Accept(Visitor);
	END_IF

END_WHILE

enumerator.Dispose();
END_METHOD

METHOD PUBLIC AddDataAsMetadata : I_Metadata
VAR_INPUT
	Name : T_MAXSTRING;
	Data : I_Datatype;
END_VAR
VAR
	metadata : I_Metadata;
END_VAR
metadata := CreateMetadata(Name, Data);
selfCreatedMetadata.Push(metadata);
AddDataAsMetadata := metadata;
END_METHOD

METHOD PUBLIC AddMetadata
VAR_INPUT
	Metadata : I_Metadata;
END_VAR
meta.AddOrUpdate(Metadata.Name, Metadata);
EmitOnMetadataAddedEvent(Metadata);
END_METHOD

PROPERTY PUBLIC HasMetadata : BOOL
GET
HasMetadata := meta.Count > 0;
END_GET
END_PROPERTY

METHOD PUBLIC SerializeWith
VAR_INPUT
	Serializer : I_Serializer;
END_VAR
VAR
	enumerator : I_ForwardEnumerator;
	metadata : I_Metadata;
END_VAR
IF meta.Count = 0 THEN
	RETURN;
END_IF

Serializer.AddKey('metadata');
Serializer.StartArray();

enumerator := meta.GetEnumerator();

WHILE enumerator.MoveNext() DO
	IF enumerator.TryGet(metadata) THEN
		metadata.SerializeWith(Serializer);
	END_IF
END_WHILE

Serializer.EndArray();
enumerator.Dispose();
END_METHOD

METHOD PUBLIC TryGetMetadataByName : BOOL
VAR_INPUT
	Name : T_MAXSTRING;
	Destination : REFERENCE TO I_Metadata;
END_VAR
VAR
	metadata : I_Metadata;
END_VAR
IF NOT meta.TryGetValue(Name, metadata) THEN
	RETURN;
END_IF

Destination := metadata;
TryGetMetadataByName := TRUE;
END_METHOD

END_FUNCTION_BLOCK

// Metadata/Events/MetadataAddedEvent
{attribute 'linkalways'} 
{attribute 'no_explicit_call' := 'This FB is a CLASS and must be accessed using methods or properties'}
{attribute 'enable_dynamic_creation'}
FUNCTION_BLOCK MetadataAddedEvent EXTENDS Disposable IMPLEMENTS I_MetadataAddedEvent
VAR
	_target : I_Metadata;
END_VAR

METHOD FB_init : BOOL
VAR_INPUT
	bInitRetains : BOOL; // if TRUE, the retain variables are initialized (warm start / cold start)
	bInCopyCode : BOOL;  // if TRUE, the instance afterwards gets moved into the copy code (online change)
	Target : I_Metadata;
END_VAR
This^._target := Target;
END_METHOD

PROPERTY PUBLIC Target : I_Metadata
GET
Target := _target;
END_GET
END_PROPERTY

END_FUNCTION_BLOCK

// Metadata/Events/I_MetadataAddedEvent
INTERFACE I_MetadataAddedEvent EXTENDS I_Event

PROPERTY PUBLIC Target : I_Metadata
GET
END_GET
END_PROPERTY

END_INTERFACE

// InputPort/Interface/I_HostInputPorts
INTERFACE I_HostInputPorts EXTENDS __SYSTEM.IQueryInterface

PROPERTY InputPorts : I_InputPorts
GET
END_GET
END_PROPERTY

END_INTERFACE

// InputPort/Interface/I_InputPorts
INTERFACE I_InputPorts

METHOD PUBLIC Accept
VAR_INPUT
	Visitor : I_InputPortVisitor;
END_VAR
END_METHOD

METHOD PUBLIC AddDataAsInputPort : I_InputPort
VAR_INPUT
	Name : T_MAXSTRING;
	Data : I_Datatype;
END_VAR
END_METHOD

METHOD AddInputPort
VAR_INPUT
	InputPort : I_InputPort;
END_VAR
END_METHOD

PROPERTY PUBLIC HasInputPorts : BOOL
GET
END_GET
END_PROPERTY

METHOD PUBLIC TryGetInputPortByName : BOOL
VAR_INPUT
	Name : T_MAXSTRING;
	Destination : REFERENCE TO I_InputPort;
END_VAR
END_METHOD

END_INTERFACE

// Visitors/Interfaces/I_InputPortVisitor
INTERFACE I_InputPortVisitor

METHOD VisitInputPort
VAR_INPUT
	VisitingInputPort : I_InputPort;
END_VAR
END_METHOD

END_INTERFACE

// InputPort/Interface/I_InputPort
INTERFACE I_InputPort EXTENDS I_Disposable, I_EventEmitter, I_EventHandler, I_Serializable, I_HostMetadata

METHOD PUBLIC Accept
VAR_INPUT
	Visitor : I_InputPortVisitor;
END_VAR
END_METHOD

PROPERTY PUBLIC Connected : BOOL
GET
END_GET
END_PROPERTY

PROPERTY PUBLIC Data : I_Datatype
GET
END_GET
END_PROPERTY

METHOD PUBLIC Disconnect
END_METHOD

PROPERTY PUBLIC Name : T_MAXSTRING
GET
END_GET
END_PROPERTY

METHOD PUBLIC TryConnectTo : BOOL
VAR_INPUT
	OutputPort : I_OutputPort;
END_VAR
END_METHOD

END_INTERFACE

// OutputPort/Base/OutputPort
{attribute 'linkalways'} 
{attribute 'no_explicit_call' := 'This FB is a CLASS and must be accessed using methods or properties'}
{attribute 'enable_dynamic_creation'}
FUNCTION_BLOCK OutputPort EXTENDS Disposable IMPLEMENTS I_OutputPort
VAR
	_name : T_MAXSTRING;
	_data : I_Datatype;
	parent : I_HostOutputPorts;
	eventEmitter : EventEmitter;
	metadataHost : MetadataHost(THIS^, eventEmitter);
END_VAR

METHOD FB_init : BOOL
VAR_INPUT
	bInitRetains : BOOL; // if TRUE, the retain variables are initialized (warm start / cold start)
	bInCopyCode : BOOL;  // if TRUE, the instance afterwards gets moved into the copy code (online change)
	Name : T_MAXSTRING;
	Data : I_Datatype;
	Parent : I_HostOutputPorts;
END_VAR
_name := Name;
_data := Data;
RegisterWithParent(Parent);
END_METHOD

METHOD Protected EmitOnOutputPortChangeEvent
VAR_INPUT
	PortChanged : I_OutputPort;
END_VAR
VAR
	pOutputPortChangeEvent : POINTER TO OutputPortChangedEvent;
END_VAR
pOutputPortChangeEvent := __NEW(OutputPortChangedEvent(Target := PortChanged));
eventEmitter.Emit('OnOutputPortChanged',pOutputPortChangeEvent^);
pOutputPortChangeEvent^.Dispose();
END_METHOD

METHOD PUBLIC Accept
VAR_INPUT
	Visitor : I_OutputPortVisitor;
END_VAR
Visitor.VisitOutputPort(THIS^);
END_METHOD

METHOD PUBLIC AddMetadata : I_HostMetadata
VAR_INPUT
	Name : T_MAXSTRING;
	Data : I_Datatype;
END_VAR
Metadatum.AddDataAsMetadata(Name, Data);
AddMetadata := THIS^;
END_METHOD

PROPERTY PUBLIC Data : I_Datatype
GET
Data := _data;
END_GET
END_PROPERTY

PROPERTY PUBLIC Metadatum : I_Metadatum
GET
Metadatum := metadataHost;
END_GET
END_PROPERTY

PROPERTY PUBLIC Name : T_MAXSTRING
GET
Name := _name;
END_GET
END_PROPERTY

METHOD PUBLIC OffEvent
VAR_INPUT
	EventName : T_MaxString;
	EventHandler : I_EventHandler;
END_VAR
eventEmitter.OffEvent(EventName, EventHandler);
END_METHOD

METHOD PUBLIC OnceEvent
VAR_INPUT
	EventName : T_MaxString;
	EventHandler : I_EventHandler;
END_VAR
eventEmitter.OnceEvent(EventName, EventHandler);
END_METHOD

METHOD PUBLIC OnEvent
VAR_INPUT
	EventName : T_MaxString;
	EventHandler : I_EventHandler;
END_VAR
eventEmitter.OnEvent(EventName, EventHandler);
END_METHOD

METHOD PUBLIC RegisterWithParent
VAR_INPUT
	Parent : I_HostOutputPorts;
END_VAR
IF Parent = 0 THEN
	RETURN;
END_IF

THIS^.parent := Parent;
Parent.OutputPorts.AddOutputPort(THIS^);
END_METHOD

METHOD PUBLIC SerializeWith
VAR_INPUT
	Serializer : I_Serializer;
END_VAR
Serializer.StartObject();
Serializer.AddKeyString('name',_name);
Serializer.Addkey('datatype');
_data.SerializeTypeWith(Serializer);
Serializer.AddkeyObject('value',_data);
metadataHost.SerializeWith(Serializer);
Serializer.EndObject();
END_METHOD

END_FUNCTION_BLOCK

// OutputPort/Interface/I_OutputPort
INTERFACE I_OutputPort EXTENDS I_Disposable, I_EventEmitter, I_Serializable, I_HostMetadata

METHOD PUBLIC Accept
VAR_INPUT
	Visitor : I_OutputPortVisitor;
END_VAR
END_METHOD

PROPERTY PUBLIC Data : I_Datatype
GET
END_GET
END_PROPERTY

PROPERTY PUBLIC Name : T_MAXSTRING
GET
END_GET
END_PROPERTY

END_INTERFACE

// Visitors/Interfaces/I_OutputPortVisitor
INTERFACE I_OutputPortVisitor

METHOD VisitOutputPort
VAR_INPUT
	VisitingOutputPort : I_OutputPort;
END_VAR
END_METHOD

END_INTERFACE

// OutputPort/Interface/I_HostOutputPorts
INTERFACE I_HostOutputPorts EXTENDS __SYSTEM.IQueryInterface

PROPERTY OutputPorts : I_OutputPorts
GET
END_GET
END_PROPERTY

END_INTERFACE

// OutputPort/Interface/I_OutputPorts
INTERFACE I_OutputPorts

METHOD PUBLIC Accept
VAR_INPUT
	Visitor : I_OutputPortVisitor;
END_VAR
END_METHOD

METHOD PUBLIC AddDataAsOutputPort : I_OutputPort
VAR_INPUT
	Name : T_MAXSTRING;
	Data : I_Datatype;
END_VAR
END_METHOD

METHOD AddOutputPort
VAR_INPUT
	OutputPort : I_OutputPort;
END_VAR
END_METHOD

PROPERTY PUBLIC HasOutputPorts : BOOL
GET
END_GET
END_PROPERTY

METHOD PUBLIC TryGetOutputPortByName : BOOL
VAR_INPUT
	Name : T_MAXSTRING;
	Destination : REFERENCE TO I_OutputPort;
END_VAR
END_METHOD

END_INTERFACE

// OutputPort/Events/OutputPortChangedEvent
{attribute 'linkalways'} 
{attribute 'no_explicit_call' := 'This FB is a CLASS and must be accessed using methods or properties'}
{attribute 'enable_dynamic_creation'}
FUNCTION_BLOCK OutputPortChangedEvent EXTENDS Disposable IMPLEMENTS I_OutputPortChangedEvent
VAR
	_target : I_OutputPort;
END_VAR

METHOD FB_init : BOOL
VAR_INPUT
	bInitRetains : BOOL; // if TRUE, the retain variables are initialized (warm start / cold start)
	bInCopyCode : BOOL;  // if TRUE, the instance afterwards gets moved into the copy code (online change)
	Target : I_OutputPort;
END_VAR
This^._target := Target;
END_METHOD

PROPERTY PUBLIC Target : I_OutputPort
GET
Target := _target;
END_GET
END_PROPERTY

END_FUNCTION_BLOCK

// OutputPort/Events/I_OutputPortChangedEvent
INTERFACE I_OutputPortChangedEvent extends I_Event

PROPERTY PUBLIC Target : I_OutputPort
GET
END_GET
END_PROPERTY

END_INTERFACE

// InputPort/Base/InputPort
{attribute 'linkalways'} 
{attribute 'no_explicit_call' := 'This FB is a CLASS and must be accessed using methods or properties'}
{attribute 'enable_dynamic_creation'}
FUNCTION_BLOCK InputPort EXTENDS Disposable IMPLEMENTS I_InputPort
VAR
	_name : T_MAXSTRING;
	_data : I_Datatype;
	_connectedTo : I_OutputPort;
	parent : I_HostInputPorts;
	eventEmitter : EventEmitter;
	metadataHost : MetadataHost(THIS^, eventEmitter);
END_VAR

METHOD FB_init : BOOL
VAR_INPUT
	bInitRetains : BOOL; // if TRUE, the retain variables are initialized (warm start / cold start)
	bInCopyCode : BOOL;  // if TRUE, the instance afterwards gets moved into the copy code (online change)
	Name : T_MAXSTRING;
	Data : I_Datatype;
	Parent : I_HostInputPorts;
END_VAR
_name := Name;
_data := Data;
RegisterWithParent(Parent);
END_METHOD

METHOD PROTECTED EmitOnInputPortChanged
VAR_INPUT
	PortChanged : I_InputPort;
END_VAR
VAR
	pInputPortChangeEvent : POINTER TO InputPortChangedEvent;
END_VAR
pInputPortChangeEvent := __NEW(InputPortChangedEvent(Target := PortChanged));
eventEmitter.Emit('OnInputPortChanged',pInputPortChangeEvent^);
pInputPortChangeEvent^.Dispose();
END_METHOD

METHOD PROTECTED HandleOutputPortChangedEvent
VAR_INPUT
	Source : I_OutputPort;
END_VAR
EmitOnInputPortChanged(THIS^);
END_METHOD

METHOD PUBLIC Accept
VAR_INPUT
	Visitor : I_InputPortVisitor;
END_VAR
Visitor.VisitInputPort(THIS^);
END_METHOD

METHOD PUBLIC AddMetadata : I_HostMetadata
VAR_INPUT
	Name : T_MAXSTRING;
	Data : I_Datatype;
END_VAR
Metadatum.AddDataAsMetadata(Name, Data);
AddMetadata := THIS^;
END_METHOD

PROPERTY PUBLIC Connected : BOOL
GET
Connected := _connectedTo <> 0;
END_GET
END_PROPERTY

PROPERTY PUBLIC Data : I_Datatype
GET
Data := _data;
END_GET
END_PROPERTY

METHOD PUBLIC Disconnect
IF NOT Connected THEN
	RETURN;
END_IF

_connectedTo.OffEvent('OnOutputPortChanged', THIS^);
_connectedTo := 0;
_data.ClearReference();
END_METHOD

METHOD PUBLIC HandleEvent
VAR_INPUT
	Event : I_Event;
END_VAR
VAR
	outputPortChangedEvent : I_OutputPortChangedEvent;
END_VAR
IF __QUERYINTERFACE(Event, outputPortChangedEvent) THEN
	HandleOutputPortChangedEvent(outputPortChangedEvent.Target);
END_IF
END_METHOD

PROPERTY PUBLIC Metadatum : I_Metadatum
GET
Metadatum := metadataHost;
END_GET
END_PROPERTY

PROPERTY PUBLIC Name : T_MAXSTRING
GET
Name := _name;
END_GET
END_PROPERTY

METHOD PUBLIC OffEvent
VAR_INPUT
	EventName : T_MaxString;
	EventHandler : I_EventHandler;
END_VAR
eventEmitter.OffEvent(EventName, EventHandler);
END_METHOD

METHOD PUBLIC OnceEvent
VAR_INPUT
	EventName : T_MaxString;
	EventHandler : I_EventHandler;
END_VAR
eventEmitter.OnceEvent(EventName, EventHandler);
END_METHOD

METHOD PUBLIC OnEvent
VAR_INPUT
	EventName : T_MaxString;
	EventHandler : I_EventHandler;
END_VAR
eventEmitter.OnEvent(EventName, EventHandler);
END_METHOD

METHOD PUBLIC RegisterWithParent
VAR_INPUT
	Parent : I_HostInputPorts;
END_VAR
IF Parent = 0 THEN
	RETURN;
END_IF

THIS^.parent := Parent;
Parent.InputPorts.AddInputPort(THIS^);
END_METHOD

METHOD PUBLIC SerializeWith
VAR_INPUT
	Serializer : I_Serializer;
END_VAR
VAR 
	isConnected : BOOL := Connected;
END_VAR
Serializer.StartObject();
Serializer.AddKeyString('name',_name);
Serializer.AddKeyBool('connected',isConnected);
Serializer.Addkey('datatype');
_data.SerializeTypeWith(Serializer);
Serializer.AddkeyObject('value',_data);
metadataHost.SerializeWith(Serializer);
Serializer.EndObject();
END_METHOD

METHOD PUBLIC TryConnectTo : BOOL
VAR_INPUT
	OutputPort : I_OutputPort;
END_VAR
IF NOT _data.TryMakeReferenceTo(OutputPort.Data) THEN
	RETURN;
END_IF

_connectedTo := OutputPort;
_connectedTo.OnEvent('OnOutputPortChanged', THIS^);
TryConnectTo := TRUE;
END_METHOD

END_FUNCTION_BLOCK

// InputPort/Events/InputPortChangedEvent
{attribute 'linkalways'} 
{attribute 'no_explicit_call' := 'This FB is a CLASS and must be accessed using methods or properties'}
{attribute 'enable_dynamic_creation'}
FUNCTION_BLOCK InputPortChangedEvent EXTENDS Disposable IMPLEMENTS I_InputPortChangedEvent
VAR
	_target : I_InputPort;
END_VAR

METHOD FB_init : BOOL
VAR_INPUT
	bInitRetains : BOOL; // if TRUE, the retain variables are initialized (warm start / cold start)
	bInCopyCode : BOOL;  // if TRUE, the instance afterwards gets moved into the copy code (online change)
	Target : I_InputPort;
END_VAR
This^._target := Target;
END_METHOD

PROPERTY PUBLIC Target : I_InputPort
GET
Target := _target;
END_GET
END_PROPERTY

END_FUNCTION_BLOCK

// InputPort/Events/I_InputPortChangedEvent
INTERFACE I_InputPortChangedEvent EXTENDS I_Event

PROPERTY PUBLIC Target : I_InputPort
GET
END_GET
END_PROPERTY

END_INTERFACE

// Parameters/Interface/I_HostParameters
INTERFACE I_HostParameters EXTENDS __SYSTEM.IQueryInterface

PROPERTY Parameters : I_Parameters
GET
END_GET
END_PROPERTY

END_INTERFACE

// Parameters/Interface/I_Parameters
INTERFACE I_Parameters

METHOD PUBLIC Accept
VAR_INPUT
	Visitor : I_ParameterVisitor;
END_VAR
END_METHOD

METHOD PUBLIC AddDataAsParameter : I_Parameter
VAR_INPUT
	Name : T_MAXSTRING;
	Data : I_Datatype;
END_VAR
END_METHOD

METHOD AddParameter
VAR_INPUT
	Parameter : I_Parameter;
END_VAR
END_METHOD

PROPERTY PUBLIC HasParameters : BOOL
GET
END_GET
END_PROPERTY

METHOD PUBLIC TryGetParameterByName : BOOL
VAR_INPUT
	Name : T_MAXSTRING;
	Destination : REFERENCE TO I_Parameter;
END_VAR
END_METHOD

END_INTERFACE

// Visitors/Interfaces/I_ParameterVisitor
INTERFACE I_ParameterVisitor

METHOD VisitParameter
VAR_INPUT
	VisitingProperty : I_Parameter;
END_VAR
END_METHOD

END_INTERFACE

// Parameters/Interface/I_Parameter
INTERFACE I_Parameter EXTENDS I_Disposable, I_Serializable, I_Deserializable, I_EventEmitter, I_HostMetadata

METHOD PUBLIC Accept
VAR_INPUT
	Visitor : I_ParameterVisitor;
END_VAR
END_METHOD

PROPERTY PUBLIC Data : I_DataType
GET
END_GET
END_PROPERTY

PROPERTY PUBLIC Name : T_MAXSTRING
GET
END_GET
END_PROPERTY

PROPERTY PUBLIC Parent : I_HostParameters
GET
END_GET
END_PROPERTY

END_INTERFACE

// Parameters/Base/Parameter
{attribute 'linkalways'} 
{attribute 'no_explicit_call' := 'This FB is a CLASS and must be accessed using methods or properties'}
{attribute 'enable_dynamic_creation'}
FUNCTION_BLOCK Parameter EXTENDS Disposable IMPLEMENTS I_Parameter
VAR
	_name : T_MAXSTRING;
	_data : I_Datatype;
	_parent : I_HostParameters;
	eventEmitter : EventEmitter;
	metadataHost : MetadataHost(THIS^, eventEmitter);
END_VAR

METHOD FB_init : BOOL
VAR_INPUT
	bInitRetains : BOOL; // if TRUE, the retain variables are initialized (warm start / cold start)
	bInCopyCode : BOOL;  // if TRUE, the instance afterwards gets moved into the copy code (online change)
	Name : T_MAXSTRING;
	Data : I_Datatype;
	Parent : I_HostParameters;
END_VAR
_name := Name;
_data := Data;
RegisterWithParent(Parent);
END_METHOD

METHOD PUBLIC Accept
VAR_INPUT
	Visitor : I_ParameterVisitor;
END_VAR
Visitor.VisitParameter(THIS^);
END_METHOD

METHOD PUBLIC AddMetadata : I_HostMetadata
VAR_INPUT
	Name : T_MAXSTRING;
	Data : I_Datatype;
END_VAR
Metadatum.AddDataAsMetadata(Name, Data);
AddMetadata := THIS^;
END_METHOD

PROPERTY PUBLIC Data : I_Datatype
GET
Data := _data;
END_GET
END_PROPERTY

PROPERTY PUBLIC Metadatum : I_Metadatum
GET
Metadatum := metadataHost;
END_GET
END_PROPERTY

PROPERTY PUBLIC Name : T_MAXSTRING
GET
Name := _name;
END_GET
END_PROPERTY

METHOD PUBLIC OffEvent
VAR_INPUT
	EventName : T_MaxString;
	EventHandler : I_EventHandler;
END_VAR
eventEmitter.OffEvent(EventName, EventHandler);
END_METHOD

METHOD PUBLIC OnceEvent
VAR_INPUT
	EventName : T_MaxString;
	EventHandler : I_EventHandler;
END_VAR
eventEmitter.OnceEvent(EventName, EventHandler);
END_METHOD

METHOD PUBLIC OnEvent
VAR_INPUT
	EventName : T_MaxString;
	EventHandler : I_EventHandler;
END_VAR
eventEmitter.OnEvent(EventName, EventHandler);
END_METHOD

PROPERTY PUBLIC Parent : I_HostParameters
GET
Parent := _parent;
END_GET
END_PROPERTY

METHOD PUBLIC RegisterWithParent
VAR_INPUT
	Parent : I_HostParameters;
END_VAR
IF Parent = 0 THEN
	RETURN;
END_IF

THIS^._parent := Parent;
Parent.Parameters.AddParameter(THIS^);
END_METHOD

METHOD PUBLIC SerializeWith
VAR_INPUT
	Serializer : I_Serializer;
END_VAR
Serializer.StartObject();
Serializer.AddKeyString('name',_name);
Serializer.Addkey('datatype');
_data.SerializeTypeWith(Serializer);
Serializer.AddkeyObject('value',_data);
metadataHost.SerializeWith(Serializer);
Serializer.EndObject();
END_METHOD

METHOD PUBLIC TryDeserializeFrom : BOOL
VAR_INPUT
	Deserializer : I_Deserializer;
	Feedback : I_DeserializerFeedback;
END_VAR
VAR
	parameterDeserializer : I_Deserializer;
END_VAR
TryDeserializeFrom := _data.TryDeserializeFrom(Deserializer, Feedback);
END_METHOD

END_FUNCTION_BLOCK

// Extensions/Interface/I_HostExtensions
INTERFACE I_HostExtensions EXTENDS __SYSTEM.IQueryInterface

PROPERTY Extensions : I_Extensions
GET
END_GET
END_PROPERTY

END_INTERFACE

// Extensions/Interface/I_Extensions
INTERFACE I_Extensions

METHOD PUBLIC Accept
VAR_INPUT
	Visitor : I_ExtensionVisitor;
END_VAR
END_METHOD

METHOD AddExtension
VAR_INPUT
	Extension : I_Extension;
END_VAR
END_METHOD

PROPERTY PUBLIC HasExtensions : BOOL
GET
END_GET
END_PROPERTY

METHOD PUBLIC TryGetExtensionByName : BOOL
VAR_INPUT
	Name : T_MAXSTRING;
	Destination : REFERENCE TO I_Extension;
END_VAR
END_METHOD

END_INTERFACE

// Visitors/Interfaces/I_ExtensionVisitor
INTERFACE I_ExtensionVisitor

METHOD VisitExtension
VAR_INPUT
	VisitingExtension : I_Extension;
END_VAR
END_METHOD

END_INTERFACE

// Extensions/Interface/I_Extension
INTERFACE I_Extension EXTENDS I_Disposable, I_HostContent, I_HostInputPorts, I_HostOutputPorts, I_HostAlarms, I_HostParameters, I_HostMetadata, I_EventEmitter, I_Deserializable, I_Serializable

METHOD PUBLIC Accept
VAR_INPUT
	Visitor : I_ExtensionVisitor;
END_VAR
END_METHOD

PROPERTY PUBLIC Name : T_MAXSTRING
GET
END_GET
END_PROPERTY

END_INTERFACE

// Extensions/Base/Extension
{attribute 'linkalways'} 
{attribute 'no_explicit_call' := 'This FB is a CLASS and must be accessed using methods or properties'}
{attribute 'enable_dynamic_creation'}
FUNCTION_BLOCK Extension EXTENDS Disposable IMPLEMENTS I_Extension
VAR
	_name : T_MAXSTRING;
	eventEmitter : EventEmitter;
	inputPortHost : InputPortHost(THIS^, eventEmitter);
	outputPortHost : OutputPortHost(THIS^, eventEmitter);
	parameterHost : ParameterHost(THIS^, eventEmitter);
	contentHost : ContentHost(THIS^, eventEmitter);
	alarmHost : AlarmHost(THIS^, eventEmitter);
	metadataHost : MetadataHost(THIS^, eventEmitter);
	deserializationFailedAlarm : DeserializationFailedAlarm(THIS^);
END_VAR

METHOD FB_init : BOOL
VAR_INPUT
	bInitRetains : BOOL; // if TRUE, the retain variables are initialized (warm start / cold start)
	bInCopyCode : BOOL;  // if TRUE, the instance afterwards gets moved into the copy code (online change)
	Name : T_MAXSTRING;
END_VAR
_name := Name;
END_METHOD

METHOD PUBLIC Accept
VAR_INPUT
	Visitor : I_ExtensionVisitor;
END_VAR
Visitor.VisitExtension(THIS^);
END_METHOD

METHOD PUBLIC AddMetadata : I_HostMetadata
VAR_INPUT
	Name : T_MAXSTRING;
	Data : I_Datatype;
END_VAR
Metadatum.AddDataAsMetadata(Name, Data);
AddMetadata := THIS^;
END_METHOD

PROPERTY PUBLIC Alarms : I_Alarms
GET
Alarms := alarmHost;
END_GET
END_PROPERTY

PROPERTY PUBLIC Contents : I_Contents
GET
Contents := contentHost;
END_GET
END_PROPERTY

PROPERTY PUBLIC HasRaisedAlarm : BOOL
GET
HasRaisedAlarm := alarmHost.HasRaisedAlarm;
END_GET
END_PROPERTY

PROPERTY PUBLIC InputPorts : I_InputPorts
GET
InputPorts := inputPortHost;
END_GET
END_PROPERTY

PROPERTY PUBLIC Metadatum : I_Metadatum
GET
Metadatum := metadataHost;
END_GET
END_PROPERTY

PROPERTY PUBLIC Name : T_MAXSTRING
GET
Name := _name;
END_GET
END_PROPERTY

METHOD PUBLIC OffEvent
VAR_INPUT
	EventName : T_MaxString;
	EventHandler : I_EventHandler;
END_VAR
eventEmitter.OffEvent(EventName, EventHandler);
END_METHOD

METHOD PUBLIC OnceEvent
VAR_INPUT
	EventName : T_MaxString;
	EventHandler : I_EventHandler;
END_VAR
eventEmitter.OnceEvent(EventName, EventHandler);
END_METHOD

METHOD PUBLIC OnEvent
VAR_INPUT
	EventName : T_MaxString;
	EventHandler : I_EventHandler;
END_VAR
eventEmitter.OnEvent(EventName, EventHandler);
END_METHOD

PROPERTY PUBLIC OutputPorts : I_OutputPorts
GET
OutputPorts := outputPortHost;
END_GET
END_PROPERTY

PROPERTY PUBLIC Parameters : I_Parameters
GET
Parameters := parameterHost;
END_GET
END_PROPERTY

METHOD PUBLIC SerializeWith
VAR_INPUT
	Serializer : I_Serializer;
END_VAR
Serializer.StartObject();
Serializer.AddKeyString('name',_name);
inputPortHost.SerializeWith(Serializer);
outputPortHost.SerializeWith(Serializer);
parameterHost.SerializeWith(Serializer);
contentHost.SerializeWith(Serializer);
alarmHost.SerializeWith(Serializer);
metadataHost.SerializeWith(Serializer);
Serializer.EndObject();
END_METHOD

METHOD PUBLIC TryDeserializeFrom : BOOL
VAR_INPUT
	Deserializer : I_Deserializer;
	Feedback : I_DeserializerFeedback;
END_VAR
DeserializationFailedAlarm.Clear();

IF NOT parameterHost.TryDeserializeFrom(Deserializer, Feedback) THEN
	DeserializationFailedAlarm.Raise('Failed to deserialize parameters');
	RETURN;
END_IF

TryDeserializeFrom := TRUE;
END_METHOD

END_FUNCTION_BLOCK

// InputPort/Host/InputPortHost
{attribute 'linkalways'} 
{attribute 'no_explicit_call' := 'This FB is a CLASS and must be accessed using methods or properties'}
{attribute 'enable_dynamic_creation'}
FUNCTION_BLOCK InputPortHost IMPLEMENTS I_InputPorts, I_Serializable
VAR
	hostParent : I_HostInputPorts;
	eventTarget : I_EventTarget;
	ports : Dictionary;
	selfCreatedInputPorts : Stack;
END_VAR

METHOD FB_init : BOOL
VAR_INPUT
	bInitRetains : BOOL; // if TRUE, the retain variables are initialized (warm start / cold start)
	bInCopyCode : BOOL;  // if TRUE, the instance afterwards gets moved into the copy code (online change)
	Parent : I_HostInputPorts;
	parentEventTarget : I_EventTarget;
END_VAR
hostParent := Parent;
eventTarget := parentEventTarget;
END_METHOD

METHOD FB_exit : BOOL
VAR_INPUT
	bInCopyCode : BOOL; // if TRUE, the exit method is called for exiting an instance that is copied afterwards (online change).
END_VAR
IF bInCopyCode THEN
	RETURN;
END_IF

DisposeSelfCreatedInputPorts();
END_METHOD

METHOD PRIVATE CreateInputPort : I_InputPort
VAR_INPUT
	PortName : T_MAXSTRING;
	PortData : I_Datatype;
END_VAR
VAR
	pPort : POINTER TO InputPort;
END_VAR
pPort := __NEW(InputPort(Name := PortName, Data := PortData, Parent := hostParent));
CreateInputPort := pPort^;
END_METHOD

METHOD PRIVATE DisposeSelfCreatedInputPorts : BOOL
VAR
	port : I_InputPort;
END_VAR
WHILE selfCreatedInputPorts.TryPop(port) DO
	port.Dispose();
END_WHILE
END_METHOD

METHOD PROTECTED EmitOnPortAddedEvent
VAR_INPUT
	Port : I_InputPort;
END_VAR
VAR
	pInputPortAddedEvent : POINTER TO InputPortAddedEvent;
END_VAR
IF eventTarget = 0 THEN
	RETURN;
END_IF

pInputPortAddedEvent := __NEW(InputPortAddedEvent(Target := Port));
eventTarget.Emit('OnInputPortAdded',pInputPortAddedEvent^);
pInputPortAddedEvent^.Dispose();
END_METHOD

METHOD PUBLIC Accept
VAR_INPUT
	Visitor : I_InputPortVisitor;
END_VAR
VAR
	enumerator : I_ForwardEnumerator;
	port : I_InputPort;
END_VAR
enumerator := ports.GetEnumerator();

WHILE (enumerator.MoveNext()) DO
	
	IF enumerator.TryGet(port) THEN
		port.Accept(Visitor);
	END_IF

END_WHILE

enumerator.Dispose();
END_METHOD

METHOD PUBLIC AddDataAsInputPort : I_InputPort
VAR_INPUT
	Name : T_MAXSTRING;
	Data : I_Datatype;
END_VAR
VAR
	port : I_InputPort;
END_VAR
port := CreateInputPort(Name, Data);
selfCreatedInputPorts.Push(port);
AddDataAsInputPort := port;
END_METHOD

METHOD PUBLIC AddInputPort
VAR_INPUT
	InputPort : I_InputPort;
END_VAR
ports.AddOrUpdate(InputPort.Name, InputPort);
EmitOnPortAddedEvent(InputPort);
END_METHOD

PROPERTY PUBLIC HasInputPorts : BOOL
GET
HasInputPorts := ports.Count > 0;
END_GET
END_PROPERTY

METHOD PUBLIC SerializeWith
VAR_INPUT
	Serializer : I_Serializer;
END_VAR
VAR
	enumerator : I_ForwardEnumerator;
	port : I_InputPort;
END_VAR
IF ports.Count = 0 THEN
	RETURN;
END_IF

Serializer.AddKey('inputPorts');
Serializer.StartArray();

enumerator := ports.GetEnumerator();

WHILE enumerator.MoveNext() DO
	IF enumerator.TryGet(port) THEN
		port.SerializeWith(Serializer);
	END_IF
END_WHILE

Serializer.EndArray();
enumerator.Dispose();
END_METHOD

METHOD PUBLIC TryGetInputPortByName : BOOL
VAR_INPUT
	Name : T_MAXSTRING;
	Destination : REFERENCE TO I_InputPort;
END_VAR
VAR
	port : I_InputPort;
END_VAR
IF NOT ports.TryGetValue(Name, port) THEN
	RETURN;
END_IF

Destination := port;
TryGetInputPortByName := TRUE;
END_METHOD

END_FUNCTION_BLOCK

// InputPort/Events/InputPortAddedEvent
{attribute 'linkalways'} 
{attribute 'no_explicit_call' := 'This FB is a CLASS and must be accessed using methods or properties'}
{attribute 'enable_dynamic_creation'}
FUNCTION_BLOCK InputPortAddedEvent EXTENDS Disposable IMPLEMENTS I_InputPortAddedEvent
VAR
	_target : I_InputPort;
END_VAR

METHOD FB_init : BOOL
VAR_INPUT
	bInitRetains : BOOL; // if TRUE, the retain variables are initialized (warm start / cold start)
	bInCopyCode : BOOL;  // if TRUE, the instance afterwards gets moved into the copy code (online change)
	Target : I_InputPort;
END_VAR
This^._target := Target;
END_METHOD

PROPERTY PUBLIC Target : I_InputPort
GET
Target := _target;
END_GET
END_PROPERTY

END_FUNCTION_BLOCK

// InputPort/Events/I_InputPortAddedEvent
INTERFACE I_InputPortAddedEvent EXTENDS I_Event

PROPERTY PUBLIC Target : I_InputPort
GET
END_GET
END_PROPERTY

END_INTERFACE

// OutputPort/Host/OutputPortHost
{attribute 'linkalways'} 
{attribute 'no_explicit_call' := 'This FB is a CLASS and must be accessed using methods or properties'}
{attribute 'enable_dynamic_creation'}
FUNCTION_BLOCK OutputPortHost IMPLEMENTS I_OutputPorts, I_Serializable
VAR
	hostParent : I_HostOutputPorts;
	eventTarget : I_EventTarget;
	ports : Dictionary;
	selfCreatedOutputPorts : Stack;
END_VAR

METHOD FB_init : BOOL
VAR_INPUT
	bInitRetains : BOOL; // if TRUE, the retain variables are initialized (warm start / cold start)
	bInCopyCode : BOOL;  // if TRUE, the instance afterwards gets moved into the copy code (online change)
	Parent : I_HostOutputPorts;
	ParentEventTarget : I_EventTarget;
END_VAR
hostParent := Parent;
eventTarget := parentEventTarget;
END_METHOD

METHOD FB_exit : BOOL
VAR_INPUT
	bInCopyCode : BOOL; // if TRUE, the exit method is called for exiting an instance that is copied afterwards (online change).
END_VAR
IF bInCopyCode THEN
	RETURN;
END_IF

DisposeSelfCreatedOutputPorts();
END_METHOD

METHOD PRIVATE CreateOutputPort : I_OutputPort
VAR_INPUT
	PortName : T_MAXSTRING;
	PortData : I_Datatype;
END_VAR
VAR
	pPort : POINTER TO OutputPort;
END_VAR
pPort := __NEW(OutputPort(Name := PortName, Data := PortData, Parent := hostParent));
CreateOutputPort := pPort^;
END_METHOD

METHOD PRIVATE DisposeSelfCreatedOutputPorts : BOOL
VAR
	port : I_OutputPort;
END_VAR
WHILE selfCreatedOutputPorts.TryPop(port) DO
	port.Dispose();
END_WHILE
END_METHOD

METHOD PROTECTED EmitOnPortAddedEvent
VAR_INPUT
	Port : I_OutputPort;
END_VAR
VAR
	pOutputPortAddedEvent : POINTER TO OutputPortAddedEvent;
END_VAR
IF eventTarget = 0 THEN
	RETURN;
END_IF

pOutputPortAddedEvent := __NEW(OutputPortAddedEvent(Target := Port));
eventTarget.Emit('OnOutputPortAdded',pOutputPortAddedEvent^);
pOutputPortAddedEvent^.Dispose();
END_METHOD

METHOD PUBLIC Accept
VAR_INPUT
	Visitor : I_OutputPortVisitor;
END_VAR
VAR
	enumerator : I_ForwardEnumerator;
	port : I_OutputPort;
END_VAR
enumerator := ports.GetEnumerator();

WHILE (enumerator.MoveNext()) DO
	
	IF enumerator.TryGet(port) THEN
		port.Accept(Visitor);
	END_IF

END_WHILE

enumerator.Dispose();
END_METHOD

METHOD PUBLIC AddDataAsOutputPort : I_OutputPort
VAR_INPUT
	Name : T_MAXSTRING;
	Data : I_Datatype;
END_VAR
VAR
	port : I_OutputPort;
END_VAR
port := CreateOutputPort(Name, Data);
selfCreatedOutputPorts.Push(port);
AddDataAsOutputPort := port;
END_METHOD

METHOD PUBLIC AddOutputPort
VAR_INPUT
	OutputPort : I_OutputPort;
END_VAR
ports.AddOrUpdate(OutputPort.Name, OutputPort);
EmitOnPortAddedEvent(OutputPort);
END_METHOD

PROPERTY PUBLIC HasOutputPorts : BOOL
GET
HasOutputPorts := ports.Count > 0;
END_GET
END_PROPERTY

METHOD PUBLIC SerializeWith
VAR_INPUT
	Serializer : I_Serializer;
END_VAR
VAR
	enumerator : I_ForwardEnumerator;
	port : I_OutputPort;
END_VAR
IF ports.Count = 0 THEN
	RETURN;
END_IF

Serializer.AddKey('outputPorts');
Serializer.StartArray();

enumerator := ports.GetEnumerator();

WHILE enumerator.MoveNext() DO
	IF enumerator.TryGet(port) THEN
		port.SerializeWith(Serializer);
	END_IF
END_WHILE

Serializer.EndArray();
enumerator.Dispose();
END_METHOD

METHOD PUBLIC TryGetOutputPortByName : BOOL
VAR_INPUT
	Name : T_MAXSTRING;
	Destination : REFERENCE TO I_OutputPort;
END_VAR
VAR
	port : I_OutputPort;
END_VAR
IF NOT ports.TryGetValue(Name, port) THEN
	RETURN;
END_IF

Destination := port;
TryGetOutputPortByName := TRUE;
END_METHOD

END_FUNCTION_BLOCK

// OutputPort/Events/OutputPortAddedEvent
{attribute 'linkalways'} 
{attribute 'no_explicit_call' := 'This FB is a CLASS and must be accessed using methods or properties'}
{attribute 'enable_dynamic_creation'}
FUNCTION_BLOCK OutputPortAddedEvent EXTENDS Disposable IMPLEMENTS I_OutputPortAddedEvent
VAR
	_target : I_OutputPort;
END_VAR

METHOD FB_init : BOOL
VAR_INPUT
	bInitRetains : BOOL; // if TRUE, the retain variables are initialized (warm start / cold start)
	bInCopyCode : BOOL;  // if TRUE, the instance afterwards gets moved into the copy code (online change)
	Target : I_OutputPort;
END_VAR
This^._target := Target;
END_METHOD

PROPERTY PUBLIC Target : I_OutputPort
GET
Target := _target;
END_GET
END_PROPERTY

END_FUNCTION_BLOCK

// OutputPort/Events/I_OutputPortAddedEvent
INTERFACE I_OutputPortAddedEvent extends I_Event

PROPERTY PUBLIC Target : I_OutputPort
GET
END_GET
END_PROPERTY

END_INTERFACE

// Parameters/Host/ParameterHost
{attribute 'linkalways'} 
{attribute 'no_explicit_call' := 'This FB is a CLASS and must be accessed using methods or properties'}
{attribute 'enable_dynamic_creation'}
FUNCTION_BLOCK ParameterHost IMPLEMENTS I_Parameters, I_Serializable
VAR
	hostParent : I_HostParameters;
	eventTarget : I_EventTarget;
	parameters : Dictionary;
	selfCreatedParameters : Stack;
END_VAR

METHOD FB_init : BOOL
VAR_INPUT
	bInitRetains : BOOL; // if TRUE, the retain variables are initialized (warm start / cold start)
	bInCopyCode : BOOL;  // if TRUE, the instance afterwards gets moved into the copy code (online change)
	Parent : I_HostParameters;
	ParentEventTarget : I_EventTarget;
END_VAR
hostParent := Parent;
eventTarget := ParentEventTarget;
END_METHOD

METHOD FB_exit : BOOL
VAR_INPUT
	bInCopyCode : BOOL; // if TRUE, the exit method is called for exiting an instance that is copied afterwards (online change).
END_VAR
IF bInCopyCode THEN
	RETURN;
END_IF

DisposeSelfCreatedParameters();
END_METHOD

METHOD PRIVATE CreateParameter : I_Parameter
VAR_INPUT
	ParameterName : T_MAXSTRING;
	ParameterData : I_Datatype;
END_VAR
VAR
	pParameter : POINTER TO Parameter;
END_VAR
pParameter := __NEW(Parameter(Name := ParameterName, Data := ParameterData, Parent := hostParent));
CreateParameter := pParameter^;
END_METHOD

METHOD PRIVATE DisposeSelfCreatedParameters : BOOL
VAR
	parameter : I_Parameter;
END_VAR
WHILE selfCreatedParameters.TryPop(parameter) DO
	parameter.Dispose();
END_WHILE
END_METHOD

METHOD PROTECTED EmitOnParameterAddedEvent
VAR_INPUT
	Parameter : I_Parameter;
END_VAR
VAR
	pParameterAddedEvent : POINTER TO ParameterAddedEvent;
END_VAR
IF eventTarget = 0 THEN
	RETURN;
END_IF

pParameterAddedEvent := __NEW(ParameterAddedEvent(TargetParameter := Parameter));
eventTarget.Emit('OnParameterAdded',pParameterAddedEvent^);
pParameterAddedEvent^.Dispose();
END_METHOD

METHOD PUBLIC Accept
VAR_INPUT
	Visitor : I_ParameterVisitor;
END_VAR
VAR
	enumerator : I_ForwardEnumerator;
	parameter : I_Parameter;
END_VAR
enumerator := parameters.GetEnumerator();

WHILE (enumerator.MoveNext()) DO
	
	IF enumerator.TryGet(parameter) THEN
		parameter.Accept(Visitor);
	END_IF

END_WHILE

enumerator.Dispose();
END_METHOD

METHOD PUBLIC AddDataAsParameter : I_Parameter
VAR_INPUT
	Name : T_MAXSTRING;
	Data : I_Datatype;
END_VAR
VAR
	parameter : I_Parameter;
END_VAR
parameter := CreateParameter(Name, Data);
selfCreatedParameters.Push(parameter);
AddDataAsParameter := parameter;
END_METHOD

METHOD PUBLIC AddParameter
VAR_INPUT
	Parameter : I_Parameter;
END_VAR
parameters.AddOrUpdate(Parameter.Name, Parameter);
EmitOnParameterAddedEvent(Parameter);
END_METHOD

PROPERTY PUBLIC HasParameters : BOOL
GET
HasParameters := parameters.Count > 0;
END_GET
END_PROPERTY

METHOD PUBLIC SerializeWith
VAR_INPUT
	Serializer : I_Serializer;
END_VAR
VAR
	enumerator : I_ForwardEnumerator;
	parameter : I_Parameter;
END_VAR
IF parameters.Count = 0 THEN
	RETURN;
END_IF

Serializer.AddKey('parameters');
Serializer.StartArray();

enumerator := parameters.GetEnumerator();

WHILE enumerator.MoveNext() DO
	IF enumerator.TryGet(parameter) THEN
		parameter.SerializeWith(Serializer);
	END_IF
END_WHILE

Serializer.EndArray();
enumerator.Dispose();
END_METHOD

METHOD PUBLIC TryDeserializeFrom : BOOL
VAR_INPUT
	Deserializer : I_Deserializer;
	Feedback : I_DeserializerFeedback;
END_VAR
VAR
	parametersDeserializer : I_Deserializer;
	parametersEnumerator : I_DeserializerObjectForwardEnumerator;
	parameter : I_Parameter;
END_VAR
parametersDeserializer := Deserializer.GetKeyObject('properties');
parametersEnumerator := parametersDeserializer.GetObjectEnumerator();

WHILE parametersEnumerator.MoveNext() DO
	
	IF NOT TryGetParameterByName(parametersEnumerator.Key, parameter) THEN
		CONTINUE;
	END_IF
	
	IF NOT parameter.TryDeserializeFrom(parametersEnumerator.Current, Feedback) THEN
		RETURN;
	END_IF

END_WHILE

TryDeserializeFrom := TRUE;
parametersEnumerator.Dispose();
END_METHOD

METHOD PUBLIC TryGetParameterByName : BOOL
VAR_INPUT
	Name : T_MAXSTRING;
	Destination : REFERENCE TO I_Parameter;
END_VAR
VAR
	parameter : I_Parameter;
END_VAR
IF NOT parameters.TryGetValue(Name, parameter) THEN
	RETURN;
END_IF

Destination := parameter;
TryGetParameterByName := TRUE;
END_METHOD

END_FUNCTION_BLOCK

// Parameters/Events/ParameterAddedEvent
{attribute 'linkalways'} 
{attribute 'no_explicit_call' := 'This FB is a CLASS and must be accessed using methods or properties'}
{attribute 'enable_dynamic_creation'}
FUNCTION_BLOCK ParameterAddedEvent EXTENDS Disposable IMPLEMENTS I_ParameterAddedEvent
VAR
	_targetParameter : I_Parameter;
END_VAR

METHOD FB_init : BOOL
VAR_INPUT
	bInitRetains : BOOL; // if TRUE, the retain variables are initialized (warm start / cold start)
	bInCopyCode : BOOL;  // if TRUE, the instance afterwards gets moved into the copy code (online change)
	TargetParameter : I_Parameter;
END_VAR
This^._targetParameter := TargetParameter;
END_METHOD

PROPERTY PUBLIC TargetParameter : I_Parameter
GET
TargetParameter := _targetParameter;
END_GET
END_PROPERTY

END_FUNCTION_BLOCK

// Parameters/Events/I_ParameterAddedEvent
INTERFACE I_ParameterAddedEvent EXTENDS I_Event

PROPERTY PUBLIC TargetParameter : I_Parameter
GET
END_GET
END_PROPERTY

END_INTERFACE

// Content/Host/ContentHost
{attribute 'linkalways'} 
{attribute 'no_explicit_call' := 'This FB is a CLASS and must be accessed using methods or properties'}
{attribute 'enable_dynamic_creation'}
FUNCTION_BLOCK ContentHost IMPLEMENTS I_Contents, I_Serializable
VAR
	hostParent : I_HostContent;
	eventTarget : I_EventTarget;
	contents : Dictionary;
	selfCreatedContent : Stack;
END_VAR

METHOD FB_init : BOOL
VAR_INPUT
	bInitRetains : BOOL; // if TRUE, the retain variables are initialized (warm start / cold start)
	bInCopyCode : BOOL;  // if TRUE, the instance afterwards gets moved into the copy code (online change)
	Parent : I_HostContent;
	ParentEventTarget : I_EventTarget;
END_VAR
hostParent := Parent;
eventTarget := parentEventTarget;
END_METHOD

METHOD FB_exit : BOOL
VAR_INPUT
	bInCopyCode : BOOL; // if TRUE, the exit method is called for exiting an instance that is copied afterwards (online change).
END_VAR
IF bInCopyCode THEN
	RETURN;
END_IF

DisposeSelfCreatedContent();
END_METHOD

METHOD PRIVATE CreateContent : I_Content
VAR_INPUT
	ContentName : T_MAXSTRING;
	ContentData : I_Datatype;
END_VAR
VAR
	pContent : POINTER TO Content;
END_VAR
pContent := __NEW(Content(Name := ContentName, Data := ContentData, Parent := hostParent));
CreateContent := pContent^;
END_METHOD

METHOD PRIVATE DisposeSelfCreatedContent : BOOL
VAR
	content : I_Content;
END_VAR
WHILE selfCreatedContent.TryPop(content) DO
	content.Dispose();
END_WHILE
END_METHOD

METHOD PROTECTED EmitOnContentAddedEvent
VAR_INPUT
	Content : I_Content;
END_VAR
VAR
	pContentAddedEvent : POINTER TO ContentAddedEvent;
END_VAR
IF eventTarget = 0 THEN
	RETURN;
END_IF

pContentAddedEvent := __NEW(ContentAddedEvent(Target := Content));
eventTarget.Emit('OnContentAdded',pContentAddedEvent^);
pContentAddedEvent^.Dispose();
END_METHOD

METHOD PUBLIC Accept
VAR_INPUT
	visitor : I_ContentVisitor;
END_VAR
VAR
	enumerator : I_ForwardEnumerator;
	content : I_Content;
END_VAR
enumerator := contents.GetEnumerator();

WHILE (enumerator.MoveNext()) DO
	
	IF enumerator.TryGet(content) THEN
		content.Accept(Visitor);
	END_IF

END_WHILE

enumerator.Dispose();
END_METHOD

METHOD PUBLIC AddContent
VAR_INPUT
	Content : I_Content;
END_VAR
contents.AddOrUpdate(Content.Name, Content);
EmitOnContentAddedEvent(Content);
END_METHOD

METHOD PUBLIC AddDataAsContent : I_Content
VAR_INPUT
	Name : T_MAXSTRING;
	Data : I_Datatype;
END_VAR
VAR
	content : I_Content;
END_VAR
content := CreateContent(Name, Data);
selfCreatedContent.Push(content);
AddDataAsContent := content;
END_METHOD

PROPERTY PUBLIC HasContents : BOOL
GET
HasContents := contents.Count > 0;
END_GET
END_PROPERTY

METHOD PUBLIC SerializeWith
VAR_INPUT
	Serializer : I_Serializer;
END_VAR
VAR
	enumerator : I_ForwardEnumerator;
	content : I_Content;
END_VAR
IF contents.Count = 0 THEN
	RETURN;
END_IF

Serializer.AddKey('contents');
Serializer.StartArray();

enumerator := contents.GetEnumerator();

WHILE enumerator.MoveNext() DO
	IF enumerator.TryGet(content) THEN
		content.SerializeWith(Serializer);
	END_IF
END_WHILE

Serializer.EndArray();
enumerator.Dispose();
END_METHOD

METHOD PUBLIC TryGetContentByName : BOOL
VAR_INPUT
	Name : T_MAXSTRING;
	Destination : REFERENCE TO I_Content;
END_VAR
VAR
	content : I_Content;
END_VAR
IF NOT contents.TryGetValue(Name, content) THEN
	RETURN;
END_IF

Destination := content;
TryGetContentByName := TRUE;
END_METHOD

END_FUNCTION_BLOCK

// Content/Events/ContentAddedEvent
{attribute 'linkalways'} 
{attribute 'no_explicit_call' := 'This FB is a CLASS and must be accessed using methods or properties'}
{attribute 'enable_dynamic_creation'}
FUNCTION_BLOCK ContentAddedEvent EXTENDS Disposable IMPLEMENTS I_ContentAddedEvent
VAR
	_target : I_Content;
END_VAR

METHOD FB_init : BOOL
VAR_INPUT
	bInitRetains : BOOL; // if TRUE, the retain variables are initialized (warm start / cold start)
	bInCopyCode : BOOL;  // if TRUE, the instance afterwards gets moved into the copy code (online change)
	Target : I_Content;
END_VAR
This^._target := Target;
END_METHOD

PROPERTY PUBLIC Target : I_Content
GET
Target := _target;
END_GET
END_PROPERTY

END_FUNCTION_BLOCK

// Content/Events/I_ContentAddedEvent
INTERFACE I_ContentAddedEvent EXTENDS I_Event

PROPERTY PUBLIC Target : I_Content
GET
END_GET
END_PROPERTY

END_INTERFACE

// Visitors/Interfaces/I_NodeVisitor
INTERFACE I_NodeVisitor

METHOD VisitNode
VAR_INPUT
	VisitingNode : I_Node;
END_VAR
END_METHOD

END_INTERFACE

// Extensions/Host/ExtensionHost
{attribute 'linkalways'} 
{attribute 'no_explicit_call' := 'This FB is a CLASS and must be accessed using methods or properties'}
{attribute 'enable_dynamic_creation'}
FUNCTION_BLOCK ExtensionHost IMPLEMENTS I_Extensions, I_Serializable, I_Deserializable
VAR
	hostParent : I_HostExtensions;
	eventTarget : I_EventTarget;
	extensions : Dictionary;
END_VAR

METHOD FB_init : BOOL
VAR_INPUT
	bInitRetains : BOOL; // if TRUE, the retain variables are initialized (warm start / cold start)
	bInCopyCode : BOOL;  // if TRUE, the instance afterwards gets moved into the copy code (online change)
	Parent : I_HostExtensions;
	ParentEventTarget : I_EventTarget;
END_VAR
hostParent := Parent;
eventTarget := parentEventTarget;
END_METHOD

METHOD PROTECTED EmitOnExtensionAddedEvent
VAR_INPUT
	Extension : I_Extension;
END_VAR
VAR
	pExtensionAddedEvent : POINTER TO ExtensionAddedEvent;
END_VAR
IF eventTarget = 0 THEN
	RETURN;
END_IF

pExtensionAddedEvent := __NEW(ExtensionAddedEvent(Target := Extension));
eventTarget.Emit('OnExtensionAdded',pExtensionAddedEvent^);
pExtensionAddedEvent^.Dispose();
END_METHOD

METHOD PUBLIC Accept
VAR_INPUT
	Visitor : I_ExtensionVisitor;
END_VAR
VAR
	enumerator : I_ForwardEnumerator;
	extension : I_Extension;
END_VAR
enumerator := extensions.GetEnumerator();

WHILE (enumerator.MoveNext()) DO
	
	IF enumerator.TryGet(extension) THEN
		extension.Accept(Visitor);
	END_IF

END_WHILE

enumerator.Dispose();
END_METHOD

METHOD PUBLIC AddExtension
VAR_INPUT
	Extension : I_Extension;
END_VAR
extensions.AddOrUpdate(Extension.Name,Extension);
EmitOnExtensionAddedEvent(Extension);
END_METHOD

PROPERTY PUBLIC HasExtensions : BOOL
GET
HasExtensions := extensions.Count > 0;
END_GET
END_PROPERTY

METHOD PUBLIC SerializeWith
VAR_INPUT
	Serializer : I_Serializer;
END_VAR
VAR
	enumerator : I_ForwardEnumerator;
	extension : I_Extension;
END_VAR
IF extensions.Count = 0 THEN
	RETURN;
END_IF

Serializer.AddKey('extensions');
Serializer.StartArray();

enumerator := extensions.GetEnumerator();

WHILE enumerator.MoveNext() DO
	IF enumerator.TryGet(extension) THEN
		extension.SerializeWith(Serializer);
	END_IF
END_WHILE

Serializer.EndArray();
enumerator.Dispose();
END_METHOD

METHOD public TryDeserializeFrom : BOOL
VAR_INPUT
	Deserializer : I_Deserializer;
	Feedback : I_DeserializerFeedback;
END_VAR
VAR
	extensionsDeserializer : I_Deserializer;
	extensionsEnumerator : I_DeserializerArrayForwardEnumerator;
	extensionName : T_MAXSTRING;
	extension : I_Extension;
END_VAR
extensionsDeserializer := Deserializer.GetKeyArray('extensions');
extensionsEnumerator := extensionsDeserializer.GetArrayEnumerator();

WHILE extensionsEnumerator.MoveNext() DO
	
	IF NOT extensionsEnumerator.Current.TryGetKeyString('name', extensionName, Feedback) THEN
		CONTINUE;
	END_IF
	
	IF NOT TryGetExtensionByName(extensionName, extension) THEN
		CONTINUE;
	END_IF
	
	IF NOT extension.TryDeserializeFrom(extensionsEnumerator.Current, Feedback) THEN
		extensionsEnumerator.Dispose();
		RETURN;
	END_IF

END_WHILE

TryDeserializeFrom := TRUE;
extensionsEnumerator.Dispose();
END_METHOD

METHOD PUBLIC TryGetExtensionByName : BOOL
VAR_INPUT
	Name : T_MAXSTRING;
	Destination : REFERENCE TO I_Extension;
END_VAR
VAR
	extension : I_Extension;
END_VAR
IF NOT extensions.TryGetValue(Name, extension) THEN
	RETURN;
END_IF

Destination := extension;
TryGetExtensionByName := TRUE;
END_METHOD

END_FUNCTION_BLOCK

// Extensions/Events/ExtensionAddedEvent
{attribute 'linkalways'} 
{attribute 'no_explicit_call' := 'This FB is a CLASS and must be accessed using methods or properties'}
{attribute 'enable_dynamic_creation'}
FUNCTION_BLOCK ExtensionAddedEvent EXTENDS Disposable IMPLEMENTS I_ExtensionAddedEvent
VAR
	_target : I_Extension;
END_VAR

METHOD FB_init : BOOL
VAR_INPUT
	bInitRetains : BOOL; // if TRUE, the retain variables are initialized (warm start / cold start)
	bInCopyCode : BOOL;  // if TRUE, the instance afterwards gets moved into the copy code (online change)
	Target : I_Extension;
END_VAR
This^._target := Target;
END_METHOD

PROPERTY PUBLIC Target : I_Extension
GET
Target := _target;
END_GET
END_PROPERTY

END_FUNCTION_BLOCK

// Extensions/Events/I_ExtensionAddedEvent
INTERFACE I_ExtensionAddedEvent EXTENDS I_Event

PROPERTY PUBLIC Target : I_Extension
GET
END_GET
END_PROPERTY

END_INTERFACE

// Node/Events/NodeExecuteBeginEvent
{attribute 'linkalways'} 
{attribute 'no_explicit_call' := 'This FB is a CLASS and must be accessed using methods or properties'}
{attribute 'enable_dynamic_creation'}
FUNCTION_BLOCK NodeExecuteBeginEvent EXTENDS Disposable IMPLEMENTS I_NodeExecuteBeginEvent
VAR
	_target : I_Node;
	_cpuCounterLowBytes : UDINT;
	_cpuCounterHighBytes : UDINT;
END_VAR

METHOD FB_init : BOOL
VAR_INPUT
	bInitRetains : BOOL; // if TRUE, the retain variables are initialized (warm start / cold start)
	bInCopyCode : BOOL;  // if TRUE, the instance afterwards gets moved into the copy code (online change)
	Target : I_Node;
END_VAR
VAR
	getCount : GETCPUCOUNTER;
END_VAR
_target := Target;
getCount(cpuCntLoDW => _cpuCounterLowBytes, cpuCntHiDW => _cpuCounterHighBytes);
END_METHOD

PROPERTY PUBLIC CpuCounterHighBytes : UDINT
GET
CpuCounterHighBytes := _cpuCounterHighBytes;
END_GET
END_PROPERTY

PROPERTY PUBLIC CpuCounterLowBytes : UDINT
GET
CpuCounterLowBytes := _cpuCounterLowBytes;
END_GET
END_PROPERTY

PROPERTY PUBLIC Target : I_Node
GET
Target := _target;
END_GET
END_PROPERTY

END_FUNCTION_BLOCK

// Node/Events/I_NodeExecuteBeginEvent
INTERFACE I_NodeExecuteBeginEvent EXTENDS I_Event

PROPERTY PUBLIC Target : I_Node
GET
END_GET
END_PROPERTY

END_INTERFACE

// Node/Events/NodeExecuteEndEvent
{attribute 'linkalways'} 
{attribute 'no_explicit_call' := 'This FB is a CLASS and must be accessed using methods or properties'}
{attribute 'enable_dynamic_creation'}
FUNCTION_BLOCK NodeExecuteEndEvent EXTENDS Disposable IMPLEMENTS I_NodeExecuteEndEvent
VAR
	_target : I_Node;
	_cpuCounterLowBytes : UDINT;
	_cpuCounterHighBytes : UDINT;
END_VAR

METHOD FB_init : BOOL
VAR_INPUT
	bInitRetains : BOOL; // if TRUE, the retain variables are initialized (warm start / cold start)
	bInCopyCode : BOOL;  // if TRUE, the instance afterwards gets moved into the copy code (online change)
	Target : I_Node;
END_VAR
VAR
	getCount : GETCPUCOUNTER;
END_VAR
_target := Target;
getCount(cpuCntLoDW => _cpuCounterLowBytes, cpuCntHiDW => _cpuCounterHighBytes);
END_METHOD

PROPERTY PUBLIC CpuCounterHighBytes : UDINT
GET
CpuCounterHighBytes := _cpuCounterHighBytes;
END_GET
END_PROPERTY

PROPERTY PUBLIC CpuCounterLowBytes : UDINT
GET
CpuCounterLowBytes := _cpuCounterLowBytes;
END_GET
END_PROPERTY

PROPERTY PUBLIC Target : I_Node
GET
Target := _target;
END_GET
END_PROPERTY

END_FUNCTION_BLOCK

// Node/Events/I_NodeExecuteEndEvent
INTERFACE I_NodeExecuteEndEvent EXTENDS I_Event

PROPERTY PUBLIC Target : I_Node
GET
END_GET
END_PROPERTY

END_INTERFACE

// Node/Events/NodePreExecuteEvent
{attribute 'linkalways'} 
{attribute 'no_explicit_call' := 'This FB is a CLASS and must be accessed using methods or properties'}
{attribute 'enable_dynamic_creation'}
FUNCTION_BLOCK NodePreExecuteEvent EXTENDS Disposable IMPLEMENTS I_NodePreExecuteEvent
VAR
	_target : I_Node;
	_cancelExecute : BOOL;
END_VAR

METHOD FB_init : BOOL
VAR_INPUT
	bInitRetains : BOOL; // if TRUE, the retain variables are initialized (warm start / cold start)
	bInCopyCode : BOOL;  // if TRUE, the instance afterwards gets moved into the copy code (online change)
	Target : I_Node;
END_VAR
_target := Target;
END_METHOD

METHOD PUBLIC Cancel
VAR_INPUT
END_VAR
_cancelExecute := true;
END_METHOD

PROPERTY PUBLIC ExecuteCancelled : BOOL
GET
ExecuteCancelled := _cancelExecute;
END_GET
END_PROPERTY

PROPERTY PUBLIC Target : I_Node
GET
Target := _target;
END_GET
END_PROPERTY

END_FUNCTION_BLOCK

// Node/Events/I_NodePreExecuteEvent
INTERFACE I_NodePreExecuteEvent EXTENDS I_Event

METHOD PUBLIC Cancel
VAR_INPUT
END_VAR
END_METHOD

PROPERTY PUBLIC ExecuteCancelled : BOOL
GET
END_GET
END_PROPERTY

PROPERTY PUBLIC Target : I_Node
GET
END_GET
END_PROPERTY

END_INTERFACE

// Alarms/FunctionFailedAlarm
{attribute 'linkalways'} 
{attribute 'no_explicit_call' := 'This FB is a CLASS and must be accessed using methods or properties'}
{attribute 'enable_dynamic_creation'}
FUNCTION_BLOCK PUBLIC FunctionFailedAlarm EXTENDS Alarm
VAR
	state : (CLEARED, RAISED);
	functionName : STRING;
	hresult : HRESULT;
END_VAR

PROPERTY Active : BOOL
GET
Active := state <> CLEARED;
END_GET
END_PROPERTY

METHOD PUBLIC Clear
functionName := '';
hresult := 0;
state := CLEARED;
END_METHOD

PROPERTY Message : T_MaxString
GET
Message := 'Function failed';
END_GET
END_PROPERTY

METHOD PUBLIC Raise
VAR_INPUT
	FunctionName : STRING;
	HResult : HRESULT;
END_VAR
THIS^.functionName := FunctionName;
THIS^.hresult := HResult;
state := RAISED;
END_METHOD

PROPERTY Reason : T_MaxString
GET
VAR
	message : STRING;
	returnCode : DWORD;
	returnCodeString : STRING;
	returnCodeMsg : STRING;
END_VAR
IF state = CLEARED THEN
	RETURN;
END_IF

returnCode := DINT_TO_DWORD(hresult) AND 16#FFF;
returnCodeString := DWORD_TO_HEXSTR(returnCode, 3, FALSE);

CASE (returnCode) OF
	
	16#70A: returnCodeMsg := 'NOMEMORY';
	16#70B: returnCodeMsg := 'INVALIDPARM';
	16#70C: returnCodeMsg := 'NOTFOUND';
	16#70E: returnCodeMsg := 'INCOMPATIBLE';
	16#712: returnCodeMsg := 'INVALIDSTATE';
	16#719: returnCodeMsg := 'TIMEOUT';
	16#71A: returnCodeMsg := 'NOINTERFACE';
	16#71B: returnCodeMsg := 'INVALIDINTERFACE';
	16#71D: returnCodeMsg := 'INVALIDOBJID';
	16#734: returnCodeMsg := 'OUTOFRANGE';
	
END_CASE


message := functionName;
message := CONCAT(message,', Msg : ');
message := CONCAT(message,returnCodeMsg);
message := CONCAT(message,', Code : 16#');
message := CONCAT(message,returnCodeString);

Reason := message;
END_GET
END_PROPERTY

END_FUNCTION_BLOCK

// Errors/MissingNodePrototypeDeserializationError
{attribute 'linkalways'} 
{attribute 'no_explicit_call' := 'This FB is a CLASS and must be accessed using methods or properties'}
{attribute 'enable_dynamic_creation'}
FUNCTION_BLOCK MissingNodePrototypeDeserializationError EXTENDS Error
VAR
	nodeType : T_MAXSTRING;
END_VAR

METHOD FB_init : BOOL
VAR_INPUT
	bInitRetains : BOOL; // if TRUE, the retain variables are initialized (warm start / cold start)
	bInCopyCode : BOOL;  // if TRUE, the instance afterwards gets moved into the copy code (online change)
	MissingType : T_MAXSTRING;
END_VAR
 nodeType := MissingType;
END_METHOD

PROPERTY PUBLIC ErrorType : T_MAXSTRING
GET
ErrorType := 'MISSING_NODE_PROTOTYPE_DESERIALIZATION_ERROR';
END_GET
END_PROPERTY

PROPERTY PUBLIC Message : T_MAXSTRING
GET
Message := CONCAT('Deserialization Failed, Missing Node Prototype : ',nodeType);
END_GET
END_PROPERTY

END_FUNCTION_BLOCK

// Extensions/Namespace/ExtensionNamespace
{attribute 'linkalways'} 
{attribute 'no_explicit_call' := 'This FB is a CLASS and must be accessed using methods or properties'}
{attribute 'enable_dynamic_creation'}
FUNCTION_BLOCK ExtensionNamespace
VAR
	_extensionName : T_MAXSTRING;
	_targetName : T_MAXSTRING;
	_isExtensionPath : BOOL;
END_VAR

METHOD FB_init : BOOL
VAR_INPUT
	bInitRetains : BOOL; // if TRUE, the retain variables are initialized (warm start / cold start)
	bInCopyCode : BOOL;  // if TRUE, the instance afterwards gets moved into the copy code (online change)
	Path : T_MAXSTRING;
END_VAR
Initialize(Path);
END_METHOD

PROPERTY PUBLIC ExtensionName : T_MAXSTRING
GET
IF NOT _isExtensionPath THEN
	RETURN;
END_IF

ExtensionName := _extensionNAme;
END_GET
END_PROPERTY

METHOD PUBLIC Initialize
VAR_INPUT
	Path : T_MAXSTRING;
END_VAR
_isExtensionPath := FindAndSplitChar(
	sSeparatorChar := '.',  
	pSrcString := ADR(Path),                                  
	pLeftString := ADR(_extensionName),   
	nLeftSize := SIZEOF(_extensionName),                                  
	pRightString := ADR(_targetName), 
	nRightSize := SIZEOF(_targetName),                                
	bSearchFromRight := TRUE 
);
END_METHOD

PROPERTY PUBLIC IsExtensionPath : BOOL
GET
IsExtensionPath := _isExtensionPath;
END_GET
END_PROPERTY

PROPERTY PUBLIC TargetName : T_MAXSTRING
GET
IF NOT _isExtensionPath THEN
	RETURN;
END_IF

TargetName := _targetName;
END_GET
END_PROPERTY

END_FUNCTION_BLOCK

// Graph/Base/Graph
{attribute 'linkalways'} 
{attribute 'no_explicit_call' := 'This FB is a CLASS and must be accessed using methods or properties'}
{attribute 'enable_dynamic_creation'}
FUNCTION_BLOCK Graph EXTENDS Disposable IMPLEMENTS I_Graph
VAR
	nodeFactory : I_NodeFactory;
	_uuid : T_MAXSTRING;	
	eventEmitter : EventEmitter;
	nodeHost : NodeHost(THIS^, eventEmitter);
	inputPortHost : InputPortHost(THIS^, eventEmitter);
	outputPortHost : OutputPortHost(THIS^, eventEmitter);
	parameterHost : ParameterHost(THIS^, eventEmitter);
	contentHost : ContentHost(THIS^, eventEmitter);
	alarmHost : AlarmHost(THIS^, eventEmitter);
	metadataHost : MetadataHost(THIS^, eventEmitter);
	extensionHost : ExtensionHost(THIS^,eventEmitter);
	selfCreatedNodes : Stack;
	
	deserializationFailedAlarm : DeserializationFailedAlarm(THIS^);
	deserializationFailedNodeNotSupportedAlarm : DeserializationFailedNodeNotSupportedAlarm(THIS^);
END_VAR

METHOD FB_init : BOOL
VAR_INPUT
	bInitRetains : BOOL; // if TRUE, the retain variables are initialized (warm start / cold start)
	bInCopyCode : BOOL;  // if TRUE, the instance afterwards gets moved into the copy code (online change)
	NodeFactory : I_NodeFactory;
END_VAR
THIS^.nodeFactory := NodeFactory;
END_METHOD

METHOD FB_exit : BOOL
VAR_INPUT
	bInCopyCode : BOOL; // if TRUE, the exit method is called for exiting an instance that is copied afterwards (online change).
END_VAR
IF bInCopyCode THEN
	RETURN;
END_IF

DisposeSelfCreatedNodes();
END_METHOD

METHOD PRIVATE DisposeSelfCreatedNodes : BOOL
VAR
	node : I_Node;
END_VAR
WHILE selfCreatedNodes.TryPop(node) DO
	nodeHost.RemoveNode(node);
	node.Dispose();
END_WHILE
END_METHOD

METHOD PUBLIC TryDeserializeLinks : BOOL
VAR_INPUT
	Deserializer : I_Deserializer;
	Feedback : I_DeserializerFeedback;
END_VAR
VAR
	linksDeserializer : I_Deserializer;
	linksEnumerator : I_DeserializerArrayForwardEnumerator;
	linkDeserializer : I_Deserializer;
	sourceNodeId : T_MAXSTRING;
	sourcePortName : T_MAXSTRING;
	destinationNodeId : T_MAXSTRING;
	destinationPortName : T_MAXSTRING;
	sourceNode : I_Node;
	sourcePort : I_OutputPort;
	destinationNode : I_Node;
	destinationPort : I_InputPort;
END_VAR
linksDeserializer := Deserializer.GetKeyArray('links');
linksEnumerator := linksDeserializer.GetArrayEnumerator();

WHILE linksEnumerator.MoveNext() DO
	
	linkDeserializer := linksEnumerator.Current.GetArray();
	
	IF NOT linkDeserializer.GetElementByIndex(1).TryGetString(sourceNodeId, Feedback) THEN
		DeserializationFailedAlarm.Raise('Missing source node id from link');
		linksEnumerator.Dispose();
		RETURN;
	END_IF
	
	IF NOT linkDeserializer.GetElementByIndex(2).TryGetString(sourcePortName, Feedback) THEN
		DeserializationFailedAlarm.Raise('Missing source port name from link');
		linksEnumerator.Dispose();
		RETURN;
	END_IF
	
	IF NOT linkDeserializer.GetElementByIndex(3).TryGetString(destinationNodeId, Feedback) THEN
		DeserializationFailedAlarm.Raise('Missing destination node id from link');
		linksEnumerator.Dispose();
		RETURN;
	END_IF
	
	IF NOT linkDeserializer.GetElementByIndex(4).TryGetString(destinationPortName, Feedback) THEN
		DeserializationFailedAlarm.Raise('Missing destination port name from link');
		linksEnumerator.Dispose();
		RETURN;
	END_IF
	
	IF NOT nodeHost.TryGetNodeById(sourceNodeId, sourceNode) THEN
		DeserializationFailedAlarm.Raise('Unable to get source node when creating link');
		linksEnumerator.Dispose();
		RETURN;
	END_IF
	
	IF NOT nodeHost.TryGetNodeById(destinationNodeId, destinationNode) THEN
		DeserializationFailedAlarm.Raise('Unable to get destination node when creating link');
		linksEnumerator.Dispose();
		RETURN;
	END_IF
	
	IF NOT sourceNode.OutputPorts.TryGetOutputPortByName(sourcePortName, sourcePort) THEN
		DeserializationFailedAlarm.Raise('Unable to get source port when creating link');
		linksEnumerator.Dispose();
		RETURN;
	END_IF
	
	IF NOT destinationNode.InputPorts.TryGetInputPortByName(destinationPortName, destinationPort) THEN
		DeserializationFailedAlarm.Raise('Unable to get destination port when creating link');
		linksEnumerator.Dispose();
		RETURN;
	END_IF
	
	IF NOT destinationPort.TryConnectTo(sourcePort) THEN
		DeserializationFailedAlarm.Raise('Unable to connect source to destination when creating link');
		linksEnumerator.Dispose();
		RETURN;
	END_IF
	
END_WHILE

TryDeserializeLinks := TRUE;
linksEnumerator.Dispose();
END_METHOD

METHOD PUBLIC TryDeserializeNodes : BOOL;
VAR_INPUT
	Deserializer : I_Deserializer;
	Feedback : I_DeserializerFeedback;
END_VAR
VAR
	nodeDeserializer : I_Deserializer;
	nodesEnumerator : I_DeserializerArrayForwardEnumerator;
	nodeType : T_MAXSTRING;
	pError : POINTER TO MissingNodePrototypeDeserializationError;
	node : I_Node;
END_VAR
nodeDeserializer := Deserializer.GetKeyArray('nodes');
nodesEnumerator := nodeDeserializer.GetArrayEnumerator();

WHILE nodesEnumerator.MoveNext() DO
	
	IF NOT nodesEnumerator.Current.TryGetKeyString('type',nodeType, Feedback) THEN
		RETURN;
	END_IF
	
	IF NOT nodeFactory.TryCreateNodeByType(nodeType, node) THEN
		pError := __NEW(MissingNodePrototypeDeserializationError(MissingType := nodeType));
		Feedback.LogError(pError^);
		DeserializationFailedNodeNotSupportedAlarm.Raise(nodeType);
		nodesEnumerator.Dispose();
		RETURN;
	END_IF
	
	selfCreatedNodes.Push(node);
	
	IF NOT node.TryDeserializeFrom(nodesEnumerator.Current, Feedback) THEN
		DeserializationFailedAlarm.Raise('Node failed to deserialize');
		nodesEnumerator.Dispose();
		RETURN;
	END_IF
	
	Nodes.AddNode(node);

END_WHILE

TryDeserializeNodes := TRUE;
nodesEnumerator.Dispose();
END_METHOD

METHOD PUBLIC Accept
VAR_INPUT
	Visitor : I_GraphVisitor;
END_VAR
Visitor.VisitGraph(THIS^);
END_METHOD

METHOD PUBLIC AddMetadata : I_HostMetadata
VAR_INPUT
	Name : T_MAXSTRING;
	Data : I_Datatype;
END_VAR
Metadatum.AddDataAsMetadata(Name, Data);
AddMetadata := THIS^;
END_METHOD

PROPERTY PUBLIC Alarms : I_Alarms
GET
Alarms := alarmHost;
END_GET
END_PROPERTY

PROPERTY PUBLIC Contents : I_Contents
GET
Contents := contentHost;
END_GET
END_PROPERTY

METHOD Execute
VAR_INPUT
END_VAR
nodeHost.Execute();
END_METHOD

PROPERTY PUBLIC Extensions : I_Extensions
GET
Extensions := extensionHost;
END_GET
END_PROPERTY

PROPERTY PUBLIC HasRaisedAlarm : BOOL
GET
HasRaisedAlarm := alarmHost.HasRaisedAlarm;
END_GET
END_PROPERTY

PROPERTY PUBLIC InputPorts : I_InputPorts
GET
InputPorts := inputPortHost;
END_GET
END_PROPERTY

PROPERTY PUBLIC Metadatum : I_Metadatum
GET
Metadatum := metadataHost;
END_GET
END_PROPERTY

PROPERTY PUBLIC Nodes : I_Nodes
GET
Nodes := nodeHost;
END_GET
END_PROPERTY

METHOD PUBLIC OffEvent
VAR_INPUT
	EventName : T_MaxString;
	EventHandler : I_EventHandler;
END_VAR
eventEmitter.OffEvent(EventName, EventHandler);
END_METHOD

METHOD PUBLIC OnceEvent
VAR_INPUT
	EventName : T_MaxString;
	EventHandler : I_EventHandler;
END_VAR
eventEmitter.OnceEvent(EventName, EventHandler);
END_METHOD

METHOD PUBLIC OnEvent
VAR_INPUT
	EventName : T_MaxString;
	EventHandler : I_EventHandler;
END_VAR
eventEmitter.OnEvent(EventName, EventHandler);
END_METHOD

PROPERTY PUBLIC OutputPorts : I_OutputPorts
GET
OutputPorts := outputPortHost;
END_GET
END_PROPERTY

PROPERTY PUBLIC Parameters : I_Parameters
GET
Parameters := parameterHost;
END_GET
END_PROPERTY

METHOD PUBLIC Reset
VAR_INPUT
END_VAR
_uuid := '';
DisposeSelfCreatedNodes();
END_METHOD

METHOD PUBLIC SerializeWith
VAR_INPUT
	Serializer : I_Serializer;
END_VAR
Serializer.StartObject();
Serializer.AddKeyString('uuid',_uuid);
inputPortHost.SerializeWith(Serializer);
outputPortHost.SerializeWith(Serializer);
parameterHost.SerializeWith(Serializer);
contentHost.SerializeWith(Serializer);
alarmHost.SerializeWith(Serializer);
extensionHost.SerializeWith(Serializer);
metadataHost.SerializeWith(Serializer);
nodeHost.SerializeWith(Serializer);
Serializer.EndObject();
END_METHOD

METHOD PUBLIC TryDeserializeFrom : BOOL
VAR_INPUT
	Deserializer : I_Deserializer;
	Feedback : I_DeserializerFeedback;
END_VAR
VAR
	receivedUuid : T_MAXSTRING;
END_VAR
DeserializationFailedNodeNotSupportedAlarm.Clear();
DeserializationFailedAlarm.Clear();

IF NOT parameterHost.TryDeserializeFrom(Deserializer, Feedback) THEN
	RETURN;
END_IF

IF NOT extensionHost.TryDeserializeFrom(Deserializer, Feedback) THEN
	RETURN;
END_IF

IF NOT Deserializer.TryGetKeyString('uuid', receivedUuid, Feedback) THEN
	RETURN;
END_IF

Reset();

IF NOT TryDeserializeNodes(Deserializer, Feedback) THEN 
	RETURN;
END_IF

IF NOT TryDeserializeLinks(Deserializer, Feedback) THEN
	RETURN;
END_IF

_uuid := receivedUuid;
TryDeserializeFrom := TRUE;
END_METHOD

PROPERTY PUBLIC Uuid : T_MAXSTRING
GET
Uuid := _uuid;
END_GET
END_PROPERTY

END_FUNCTION_BLOCK

// Graph/Interfaces/I_Graph
INTERFACE I_Graph EXTENDS I_Disposable, I_HostNodes, I_HostContent, I_HostInputPorts, I_HostOutputPorts, I_HostAlarms, I_HostParameters, I_HostExtensions, I_HostMetadata, I_EventEmitter, I_Deserializable, I_Serializable

METHOD PUBLIC Accept
VAR_INPUT
	Visitor : I_GraphVisitor;
END_VAR
END_METHOD

METHOD Execute
VAR_INPUT
END_VAR
END_METHOD

METHOD PUBLIC Reset
VAR_INPUT
END_VAR
END_METHOD

PROPERTY PUBLIC Uuid : T_MAXSTRING
GET
END_GET
END_PROPERTY

END_INTERFACE

// Node/Interface/I_HostNodes
INTERFACE I_HostNodes

PROPERTY Nodes : I_Nodes
GET
END_GET
END_PROPERTY

END_INTERFACE

// Node/Interface/I_Nodes
INTERFACE I_Nodes

METHOD PUBLIC Accept
VAR_INPUT
	Visitor : I_NodeVisitor;
END_VAR
END_METHOD

METHOD AddNode
VAR_INPUT
	Node : I_Node;
END_VAR
END_METHOD

PROPERTY PUBLIC HasNodes : BOOL
GET
END_GET
END_PROPERTY

METHOD PUBLIC TryGetNodeById : BOOL
VAR_INPUT
	Id : T_MAXSTRING;
	Destination : REFERENCE TO I_Node;
END_VAR
END_METHOD

END_INTERFACE

// Visitors/Interfaces/I_GraphVisitor
INTERFACE I_GraphVisitor

METHOD VisitGraph
VAR_INPUT
	VisitingGraph : I_Graph;
END_VAR
END_METHOD

END_INTERFACE

// NodeFactory/Base/NodeFactory
{attribute 'linkalways'} 
{attribute 'no_explicit_call' := 'This FB is a CLASS and must be accessed using methods or properties'}
{attribute 'enable_dynamic_creation'}
FUNCTION_BLOCK NodeFactory IMPLEMENTS I_NodeFactory
VAR
	prototypeHost : NodePrototypeHost;
END_VAR

METHOD PUBLIC Accept
VAR_INPUT
	Visitor : I_NodeFactoryVisitor;
END_VAR
Visitor.VisitNodeFactory(this^);
END_METHOD

METHOD AddNodeAsPrototype : I_NodePrototype
VAR_INPUT
	Path : T_MAXSTRING;
	Node : I_Node;
END_VAR
AddNodeAsPrototype := prototypeHost.AddNodeAsPrototype(Path, Node);
END_METHOD

METHOD PUBLIC AddNodePrototype
VAR_INPUT
	NodePrototype : I_NodePrototype;
END_VAR
prototypeHost.AddNodePrototype(NodePrototype);
END_METHOD

PROPERTY PUBLIC NodePrototypes : I_NodePrototypes
GET
NodePrototypes := prototypeHost;
END_GET
END_PROPERTY

METHOD PUBLIC TryCreateNodeByType : BOOL
VAR_INPUT
	Path : T_MAXSTRING;
	Destination : REFERENCE TO I_Node;
END_VAR
VAR
	nodePrototype : I_NodePrototype;
END_VAR
IF NOT prototypeHost.TryGetNodePrototypeByPath(Path, nodePrototype) THEN
	RETURN;
END_IF

Destination := nodePrototype.Clone();
TryCreateNodeByType := TRUE;
END_METHOD

END_FUNCTION_BLOCK

// NodeFactory/Interface/I_NodeFactory
INTERFACE I_NodeFactory

METHOD PUBLIC Accept
VAR_INPUT
	Visitor : I_NodeFactoryVisitor;
END_VAR
END_METHOD

METHOD AddNodeAsPrototype : I_NodePrototype
VAR_INPUT
	Path : T_MAXSTRING;
	Node : I_Node;
END_VAR
END_METHOD

METHOD PUBLIC AddNodePrototype
VAR_INPUT
	NodePrototype : I_NodePrototype;
END_VAR
END_METHOD

PROPERTY PUBLIC ABSTRACT NodePrototypes : I_NodePrototypes
GET
END_GET
END_PROPERTY

METHOD PUBLIC TryCreateNodeByType : BOOL
VAR_INPUT
	Path : T_MAXSTRING;
	Destination : REFERENCE TO I_Node;
END_VAR
END_METHOD

END_INTERFACE

// Visitors/Interfaces/I_NodeFactoryVisitor
INTERFACE I_NodeFactoryVisitor

METHOD VisitNodeFactory
VAR_INPUT
	VisitingNodeFactory : I_NodeFactory;
END_VAR
END_METHOD

END_INTERFACE

// NodePrototype/Interface/I_NodePrototype
INTERFACE I_NodePrototype EXTENDS I_Disposable

METHOD PUBLIC Accept
VAR_INPUT
	Visitor : I_NodePrototypeVisitor;
END_VAR
END_METHOD

METHOD PUBLIC Clone : I_Node
VAR_INPUT
END_VAR
END_METHOD

PROPERTY PUBLIC Node : I_Node
GET
END_GET
END_PROPERTY

PROPERTY PUBLIC Path : T_MAXSTRING
GET
END_GET
END_PROPERTY

END_INTERFACE

// Visitors/Interfaces/I_NodePrototypeVisitor
INTERFACE I_NodePrototypeVisitor

METHOD VisitNodePrototype
VAR_INPUT
	VisitingPrototype : I_NodePrototype;
END_VAR
END_METHOD

END_INTERFACE

// NodePrototype/Base/NodePrototype
{attribute 'linkalways'} 
{attribute 'no_explicit_call' := 'This FB is a CLASS and must be accessed using methods or properties'}
{attribute 'enable_dynamic_creation'}
FUNCTION_BLOCK NodePrototype EXTENDS Disposable IMPLEMENTS I_NodePrototype
VAR
	_path : T_MAXSTRING;
	_node : I_Node;
END_VAR

METHOD FB_init : BOOL
VAR_INPUT
	bInitRetains : BOOL; // if TRUE, the retain variables are initialized (warm start / cold start)
	bInCopyCode : BOOL;  // if TRUE, the instance afterwards gets moved into the copy code (online change)
	Path : T_MAXSTRING;
	Node : I_Node;
END_VAR
_path := Path;
_node := Node;
END_METHOD

METHOD PUBLIC Accept
VAR_INPUT
	Visitor : I_NodePrototypeVisitor;
END_VAR
Visitor.VisitNodePrototype(This^);
END_METHOD

METHOD PUBLIC Clone : I_Node
VAR_INPUT
END_VAR
Clone := _node.Clone();
END_METHOD

PROPERTY PUBLIC Node : I_Node
GET
Node := _node;
END_GET
END_PROPERTY

PROPERTY PUBLIC Path : T_MAXSTRING
GET
Path := _path;
END_GET
END_PROPERTY

END_FUNCTION_BLOCK

// NodePrototype/Interface/I_NodePrototypes
INTERFACE I_NodePrototypes

METHOD PUBLIC Accept
VAR_INPUT
	Visitor : I_NodePrototypeVisitor;
END_VAR
END_METHOD

PROPERTY PUBLIC HasNodePrototypes : BOOL
GET
END_GET
END_PROPERTY

END_INTERFACE

// NodePrototype/Host/NodePrototypeHost
{attribute 'linkalways'} 
{attribute 'no_explicit_call' := 'This FB is a CLASS and must be accessed using methods or properties'}
{attribute 'enable_dynamic_creation'}
FUNCTION_BLOCK NodePrototypeHost IMPLEMENTS I_NodePrototypes
VAR
	prototypes : Dictionary;
	selfCreatedPrototypes : Stack;
END_VAR

METHOD FB_exit : BOOL
VAR_INPUT
	bInCopyCode : BOOL; // if TRUE, the exit method is called for exiting an instance that is copied afterwards (online change).
END_VAR
IF bInCopyCode THEN
	RETURN;
END_IF

DisposeSelfCreatedNodePrototypes();
END_METHOD

